# B&R Automation Studio project mapp6d_SampleProject
Automation Studio 4.10.2.37; technology packages: mapp6D 1.1.7924

## Configuration Config1

CPU X20CP3586, AutomationRuntime B4.91, Build 4.1.2, Safety 0.0, Vc V4.72.3

### Task classes (Cpu.sw)
```
Cyclic#4:
  Program <- Program.prg
Libraries: McAcp6D, McBase, AsMath
```

### Hardware
```
8YFLM01.0000.00I-1 : 8YFLM01.0000.00I-1 v0.0.0.1  [PLK1 -> X20CP3586.IF3 (NodeNumber=16) [Cable Type=PowerlinkCable, Length=10, Version=1.0.0.3]]
  Supervision = off
X20CP3586 : X20CP3586 v1.9.0.0
  Connector IF2:
    ActivateDevice = 1
    Mode = Manual
    InternetAddress = 192.168.10.7
    SubnetMask = 255.255.255.0
    ActivateSnmp = 2
  Connector IF3:
    CycleTime = 1000
  ConfigurationID = mapp6d_SampleProject_Config1
  TimerDeviceType = EPLX2X
  TimerDevice = X20CP3586.IF3
  TaskClassIdleTime = 2000
  Cyclic1Duration = 1000
  Cyclic1Tolerance = 0
  Cyclic3Duration = 52000
  Cyclic3Tolerance = 52000
  Cyclic5Duration = 198000
  Cyclic5Tolerance = 198000
  Cyclic7Duration = 1002000
  Cyclic7Tolerance = 1002000
  FileDevice1
  FileDeviceName1 = 6DData
  FileDevicePath1 = C:\
  FtpUser1
  FtpUsername1 = admin
  FtpUserPassword1 = lR/ROkjEB6ZsaZw8IVX3MB+yAH7U94gbA110ofjiao0=  // admin
  FtpUserSalt1 = rhukc7YS
  FTPAccessRight1 = 0
  FTPdevice1 = ALL
```

### IoMap.iom - X20CP3586/IoMap.iom
```iecst
VAR_CONFIG
	Cyclic#1.::FBin.Array[0] AT %IW."8YFLM01.0000.00I-1".EPL_FB_IN_0_I2007_S01;
	Cyclic#1.::FBin.Array[1] AT %IW."8YFLM01.0000.00I-1".EPL_FB_IN_1_I2007_S02;
	Cyclic#1.::FBin.Array[10] AT %IW."8YFLM01.0000.00I-1".EPL_FB_IN_10_I2007_S0B;
	Cyclic#1.::FBin.Array[100] AT %IW."8YFLM01.0000.00I-1".EPL_FB_IN_100_I2007_S65;
	Cyclic#1.::FBin.Array[101] AT %IW."8YFLM01.0000.00I-1".EPL_FB_IN_101_I2007_S66;
	Cyclic#1.::FBin.Array[102] AT %IW."8YFLM01.0000.00I-1".EPL_FB_IN_102_I2007_S67;
	Cyclic#1.::FBin.Array[103] AT %IW."8YFLM01.0000.00I-1".EPL_FB_IN_103_I2007_S68;
	Cyclic#1.::FBin.Array[104] AT %IW."8YFLM01.0000.00I-1".EPL_FB_IN_104_I2007_S69;
	Cyclic#1.::FBin.Array[105] AT %IW."8YFLM01.0000.00I-1".EPL_FB_IN_105_I2007_S6A;
	Cyclic#1.::FBin.Array[106] AT %IW."8YFLM01.0000.00I-1".EPL_FB_IN_106_I2007_S6B;
	Cyclic#1.::FBin.Array[107] AT %IW."8YFLM01.0000.00I-1".EPL_FB_IN_107_I2007_S6C;
	Cyclic#1.::FBin.Array[108] AT %IW."8YFLM01.0000.00I-1".EPL_FB_IN_108_I2007_S6D;
	Cyclic#1.::FBin.Array[109] AT %IW."8YFLM01.0000.00I-1".EPL_FB_IN_109_I2007_S6E;
	Cyclic#1.::FBin.Array[11] AT %IW."8YFLM01.0000.00I-1".EPL_FB_IN_11_I2007_S0C;
	Cyclic#1.::FBin.Array[110] AT %IW."8YFLM01.0000.00I-1".EPL_FB_IN_110_I2007_S6F;
	Cyclic#1.::FBin.Array[111] AT %IW."8YFLM01.0000.00I-1".EPL_FB_IN_111_I2007_S70;
	Cyclic#1.::FBin.Array[112] AT %IW."8YFLM01.0000.00I-1".EPL_FB_IN_112_I2007_S71;
	Cyclic#1.::FBin.Array[113] AT %IW."8YFLM01.0000.00I-1".EPL_FB_IN_113_I2007_S72;
	Cyclic#1.::FBin.Array[114] AT %IW."8YFLM01.0000.00I-1".EPL_FB_IN_114_I2007_S73;
	Cyclic#1.::FBin.Array[115] AT %IW."8YFLM01.0000.00I-1".EPL_FB_IN_115_I2007_S74;
	Cyclic#1.::FBin.Array[116] AT %IW."8YFLM01.0000.00I-1".EPL_FB_IN_116_I2007_S75;
	Cyclic#1.::FBin.Array[117] AT %IW."8YFLM01.0000.00I-1".EPL_FB_IN_117_I2007_S76;
	Cyclic#1.::FBin.Array[118] AT %IW."8YFLM01.0000.00I-1".EPL_FB_IN_118_I2007_S77;
	Cyclic#1.::FBin.Array[119] AT %IW."8YFLM01.0000.00I-1".EPL_FB_IN_119_I2007_S78;
	Cyclic#1.::FBin.Array[12] AT %IW."8YFLM01.0000.00I-1".EPL_FB_IN_12_I2007_S0D;
	Cyclic#1.::FBin.Array[120] AT %IW."8YFLM01.0000.00I-1".EPL_FB_IN_120_I2007_S79;
	Cyclic#1.::FBin.Array[121] AT %IW."8YFLM01.0000.00I-1".EPL_FB_IN_121_I2007_S7A;
	Cyclic#1.::FBin.Array[122] AT %IW."8YFLM01.0000.00I-1".EPL_FB_IN_122_I2007_S7B;
	Cyclic#1.::FBin.Array[123] AT %IW."8YFLM01.0000.00I-1".EPL_FB_IN_123_I2007_S7C;
	Cyclic#1.::FBin.Array[124] AT %IW."8YFLM01.0000.00I-1".EPL_FB_IN_124_I2007_S7D;
	Cyclic#1.::FBin.Array[125] AT %IW."8YFLM01.0000.00I-1".EPL_FB_IN_125_I2007_S7E;
	Cyclic#1.::FBin.Array[126] AT %IW."8YFLM01.0000.00I-1".EPL_FB_IN_126_I2007_S7F;
	Cyclic#1.::FBin.Array[127] AT %IW."8YFLM01.0000.00I-1".EPL_FB_IN_127_I2007_S80;
	Cyclic#1.::FBin.Array[128] AT %IW."8YFLM01.0000.00I-1".EPL_FB_IN_128_I2007_S81;
	Cyclic#1.::FBin.Array[129] AT %IW."8YFLM01.0000.00I-1".EPL_FB_IN_129_I2007_S82;
	Cyclic#1.::FBin.Array[13] AT %IW."8YFLM01.0000.00I-1".EPL_FB_IN_13_I2007_S0E;
	Cyclic#1.::FBin.Array[130] AT %IW."8YFLM01.0000.00I-1".EPL_FB_IN_130_I2007_S83;
	Cyclic#1.::FBin.Array[131] AT %IW."8YFLM01.0000.00I-1".EPL_FB_IN_131_I2007_S84;
	Cyclic#1.::FBin.Array[132] AT %IW."8YFLM01.0000.00I-1".EPL_FB_IN_132_I2007_S85;
	Cyclic#1.::FBin.Array[133] AT %IW."8YFLM01.0000.00I-1".EPL_FB_IN_133_I2007_S86;
	Cyclic#1.::FBin.Array[134] AT %IW."8YFLM01.0000.00I-1".EPL_FB_IN_134_I2007_S87;
	Cyclic#1.::FBin.Array[135] AT %IW."8YFLM01.0000.00I-1".EPL_FB_IN_135_I2007_S88;
	Cyclic#1.::FBin.Array[136] AT %IW."8YFLM01.0000.00I-1".EPL_FB_IN_136_I2007_S89;
	Cyclic#1.::FBin.Array[137] AT %IW."8YFLM01.0000.00I-1".EPL_FB_IN_137_I2007_S8A;
	Cyclic#1.::FBin.Array[138] AT %IW."8YFLM01.0000.00I-1".EPL_FB_IN_138_I2007_S8B;
	Cyclic#1.::FBin.Array[139] AT %IW."8YFLM01.0000.00I-1".EPL_FB_IN_139_I2007_S8C;
	Cyclic#1.::FBin.Array[14] AT %IW."8YFLM01.0000.00I-1".EPL_FB_IN_14_I2007_S0F;
	Cyclic#1.::FBin.Array[140] AT %IW."8YFLM01.0000.00I-1".EPL_FB_IN_140_I2007_S8D;
	Cyclic#1.::FBin.Array[141] AT %IW."8YFLM01.0000.00I-1".EPL_FB_IN_141_I2007_S8E;
	Cyclic#1.::FBin.Array[142] AT %IW."8YFLM01.0000.00I-1".EPL_FB_IN_142_I2007_S8F;
	Cyclic#1.::FBin.Array[143] AT %IW."8YFLM01.0000.00I-1".EPL_FB_IN_143_I2007_S90;
	Cyclic#1.::FBin.Array[144] AT %IW."8YFLM01.0000.00I-1".EPL_FB_IN_144_I2007_S91;
	Cyclic#1.::FBin.Array[145] AT %IW."8YFLM01.0000.00I-1".EPL_FB_IN_145_I2007_S92;
	Cyclic#1.::FBin.Array[146] AT %IW."8YFLM01.0000.00I-1".EPL_FB_IN_146_I2007_S93;
	Cyclic#1.::FBin.Array[147] AT %IW."8YFLM01.0000.00I-1".EPL_FB_IN_147_I2007_S94;
	Cyclic#1.::FBin.Array[148] AT %IW."8YFLM01.0000.00I-1".EPL_FB_IN_148_I2007_S95;
	Cyclic#1.::FBin.Array[149] AT %IW."8YFLM01.0000.00I-1".EPL_FB_IN_149_I2007_S96;
	Cyclic#1.::FBin.Array[15] AT %IW."8YFLM01.0000.00I-1".EPL_FB_IN_15_I2007_S10;
	Cyclic#1.::FBin.Array[150] AT %IW."8YFLM01.0000.00I-1".EPL_FB_IN_150_I2007_S97;
	Cyclic#1.::FBin.Array[151] AT %IW."8YFLM01.0000.00I-1".EPL_FB_IN_151_I2007_S98;
	Cyclic#1.::FBin.Array[152] AT %IW."8YFLM01.0000.00I-1".EPL_FB_IN_152_I2007_S99;
	Cyclic#1.::FBin.Array[153] AT %IW."8YFLM01.0000.00I-1".EPL_FB_IN_153_I2007_S9A;
	Cyclic#1.::FBin.Array[154] AT %IW."8YFLM01.0000.00I-1".EPL_FB_IN_154_I2007_S9B;
	Cyclic#1.::FBin.Array[155] AT %IW."8YFLM01.0000.00I-1".EPL_FB_IN_155_I2007_S9C;
	Cyclic#1.::FBin.Array[156] AT %IW."8YFLM01.0000.00I-1".EPL_FB_IN_156_I2007_S9D;
	Cyclic#1.::FBin.Array[157] AT %IW."8YFLM01.0000.00I-1".EPL_FB_IN_157_I2007_S9E;
	Cyclic#1.::FBin.Array[158] AT %IW."8YFLM01.0000.00I-1".EPL_FB_IN_158_I2007_S9F;
	Cyclic#1.::FBin.Array[159] AT %IW."8YFLM01.0000.00I-1".EPL_FB_IN_159_I2007_SA0;
	Cyclic#1.::FBin.Array[16] AT %IW."8YFLM01.0000.00I-1".EPL_FB_IN_16_I2007_S11;
	Cyclic#1.::FBin.Array[160] AT %IW."8YFLM01.0000.00I-1".EPL_FB_IN_160_I2007_SA1;
	Cyclic#1.::FBin.Array[161] AT %IW."8YFLM01.0000.00I-1".EPL_FB_IN_161_I2007_SA2;
	Cyclic#1.::FBin.Array[162] AT %IW."8YFLM01.0000.00I-1".EPL_FB_IN_162_I2007_SA3;
	Cyclic#1.::FBin.Array[163] AT %IW."8YFLM01.0000.00I-1".EPL_FB_IN_163_I2007_SA4;
	Cyclic#1.::FBin.Array[164] AT %IW."8YFLM01.0000.00I-1".EPL_FB_IN_164_I2007_SA5;
	Cyclic#1.::FBin.Array[165] AT %IW."8YFLM01.0000.00I-1".EPL_FB_IN_165_I2007_SA6;
	Cyclic#1.::FBin.Array[166] AT %IW."8YFLM01.0000.00I-1".EPL_FB_IN_166_I2007_SA7;
	Cyclic#1.::FBin.Array[167] AT %IW."8YFLM01.0000.00I-1".EPL_FB_IN_167_I2007_SA8;
	Cyclic#1.::FBin.Array[168] AT %IW."8YFLM01.0000.00I-1".EPL_FB_IN_168_I2007_SA9;
	Cyclic#1.::FBin.Array[169] AT %IW."8YFLM01.0000.00I-1".EPL_FB_IN_169_I2007_SAA;
	Cyclic#1.::FBin.Array[17] AT %IW."8YFLM01.0000.00I-1".EPL_FB_IN_17_I2007_S12;
	Cyclic#1.::FBin.Array[170] AT %IW."8YFLM01.0000.00I-1".EPL_FB_IN_170_I2007_SAB;
	Cyclic#1.::FBin.Array[171] AT %IW."8YFLM01.0000.00I-1".EPL_FB_IN_171_I2007_SAC;
	Cyclic#1.::FBin.Array[172] AT %IW."8YFLM01.0000.00I-1".EPL_FB_IN_172_I2007_SAD;
	Cyclic#1.::FBin.Array[173] AT %IW."8YFLM01.0000.00I-1".EPL_FB_IN_173_I2007_SAE;
	Cyclic#1.::FBin.Array[174] AT %IW."8YFLM01.0000.00I-1".EPL_FB_IN_174_I2007_SAF;
	Cyclic#1.::FBin.Array[175] AT %IW."8YFLM01.0000.00I-1".EPL_FB_IN_175_I2007_SB0;
	Cyclic#1.::FBin.Array[176] AT %IW."8YFLM01.0000.00I-1".EPL_FB_IN_176_I2007_SB1;
	Cyclic#1.::FBin.Array[177] AT %IW."8YFLM01.0000.00I-1".EPL_FB_IN_177_I2007_SB2;
	Cyclic#1.::FBin.Array[178] AT %IW."8YFLM01.0000.00I-1".EPL_FB_IN_178_I2007_SB3;
	Cyclic#1.::FBin.Array[179] AT %IW."8YFLM01.0000.00I-1".EPL_FB_IN_179_I2007_SB4;
	Cyclic#1.::FBin.Array[18] AT %IW."8YFLM01.0000.00I-1".EPL_FB_IN_18_I2007_S13;
	Cyclic#1.::FBin.Array[180] AT %IW."8YFLM01.0000.00I-1".EPL_FB_IN_180_I2007_SB5;
	Cyclic#1.::FBin.Array[181] AT %IW."8YFLM01.0000.00I-1".EPL_FB_IN_181_I2007_SB6;
	Cyclic#1.::FBin.Array[182] AT %IW."8YFLM01.0000.00I-1".EPL_FB_IN_182_I2007_SB7;
	Cyclic#1.::FBin.Array[183] AT %IW."8YFLM01.0000.00I-1".EPL_FB_IN_183_I2007_SB8;
	Cyclic#1.::FBin.Array[184] AT %IW."8YFLM01.0000.00I-1".EPL_FB_IN_184_I2007_SB9;
	Cyclic#1.::FBin.Array[185] AT %IW."8YFLM01.0000.00I-1".EPL_FB_IN_185_I2007_SBA;
	Cyclic#1.::FBin.Array[186] AT %IW."8YFLM01.0000.00I-1".EPL_FB_IN_186_I2007_SBB;
	Cyclic#1.::FBin.Array[187] AT %IW."8YFLM01.0000.00I-1".EPL_FB_IN_187_I2007_SBC;
	Cyclic#1.::FBin.Array[188] AT %IW."8YFLM01.0000.00I-1".EPL_FB_IN_188_I2007_SBD;
	Cyclic#1.::FBin.Array[189] AT %IW."8YFLM01.0000.00I-1".EPL_FB_IN_189_I2007_SBE;
	Cyclic#1.::FBin.Array[19] AT %IW."8YFLM01.0000.00I-1".EPL_FB_IN_19_I2007_S14;
	Cyclic#1.::FBin.Array[190] AT %IW."8YFLM01.0000.00I-1".EPL_FB_IN_190_I2007_SBF;
	Cyclic#1.::FBin.Array[191] AT %IW."8YFLM01.0000.00I-1".EPL_FB_IN_191_I2007_SC0;
	Cyclic#1.::FBin.Array[192] AT %IW."8YFLM01.0000.00I-1".EPL_FB_IN_192_I2007_SC1;
	Cyclic#1.::FBin.Array[193] AT %IW."8YFLM01.0000.00I-1".EPL_FB_IN_193_I2007_SC2;
	Cyclic#1.::FBin.Array[194] AT %IW."8YFLM01.0000.00I-1".EPL_FB_IN_194_I2007_SC3;
	Cyclic#1.::FBin.Array[195] AT %IW."8YFLM01.0000.00I-1".EPL_FB_IN_195_I2007_SC4;
	Cyclic#1.::FBin.Array[196] AT %IW."8YFLM01.0000.00I-1".EPL_FB_IN_196_I2007_SC5;
	Cyclic#1.::FBin.Array[197] AT %IW."8YFLM01.0000.00I-1".EPL_FB_IN_197_I2007_SC6;
	Cyclic#1.::FBin.Array[198] AT %IW."8YFLM01.0000.00I-1".EPL_FB_IN_198_I2007_SC7;
	Cyclic#1.::FBin.Array[199] AT %IW."8YFLM01.0000.00I-1".EPL_FB_IN_199_I2007_SC8;
	Cyclic#1.::FBin.Array[2] AT %IW."8YFLM01.0000.00I-1".EPL_FB_IN_2_I2007_S03;
	Cyclic#1.::FBin.Array[20] AT %IW."8YFLM01.0000.00I-1".EPL_FB_IN_20_I2007_S15;
	Cyclic#1.::FBin.Array[21] AT %IW."8YFLM01.0000.00I-1".EPL_FB_IN_21_I2007_S16;
	Cyclic#1.::FBin.Array[22] AT %IW."8YFLM01.0000.00I-1".EPL_FB_IN_22_I2007_S17;
	Cyclic#1.::FBin.Array[23] AT %IW."8YFLM01.0000.00I-1".EPL_FB_IN_23_I2007_S18;
	Cyclic#1.::FBin.Array[24] AT %IW."8YFLM01.0000.00I-1".EPL_FB_IN_24_I2007_S19;
	Cyclic#1.::FBin.Array[25] AT %IW."8YFLM01.0000.00I-1".EPL_FB_IN_25_I2007_S1A;
	Cyclic#1.::FBin.Array[26] AT %IW."8YFLM01.0000.00I-1".EPL_FB_IN_26_I2007_S1B;
	Cyclic#1.::FBin.Array[27] AT %IW."8YFLM01.0000.00I-1".EPL_FB_IN_27_I2007_S1C;
	Cyclic#1.::FBin.Array[28] AT %IW."8YFLM01.0000.00I-1".EPL_FB_IN_28_I2007_S1D;
	Cyclic#1.::FBin.Array[29] AT %IW."8YFLM01.0000.00I-1".EPL_FB_IN_29_I2007_S1E;
	Cyclic#1.::FBin.Array[3] AT %IW."8YFLM01.0000.00I-1".EPL_FB_IN_3_I2007_S04;
	Cyclic#1.::FBin.Array[30] AT %IW."8YFLM01.0000.00I-1".EPL_FB_IN_30_I2007_S1F;
	Cyclic#1.::FBin.Array[31] AT %IW."8YFLM01.0000.00I-1".EPL_FB_IN_31_I2007_S20;
	Cyclic#1.::FBin.Array[32] AT %IW."8YFLM01.0000.00I-1".EPL_FB_IN_32_I2007_S21;
	Cyclic#1.::FBin.Array[33] AT %IW."8YFLM01.0000.00I-1".EPL_FB_IN_33_I2007_S22;
	Cyclic#1.::FBin.Array[34] AT %IW."8YFLM01.0000.00I-1".EPL_FB_IN_34_I2007_S23;
	Cyclic#1.::FBin.Array[35] AT %IW."8YFLM01.0000.00I-1".EPL_FB_IN_35_I2007_S24;
	Cyclic#1.::FBin.Array[36] AT %IW."8YFLM01.0000.00I-1".EPL_FB_IN_36_I2007_S25;
	Cyclic#1.::FBin.Array[37] AT %IW."8YFLM01.0000.00I-1".EPL_FB_IN_37_I2007_S26;
	Cyclic#1.::FBin.Array[38] AT %IW."8YFLM01.0000.00I-1".EPL_FB_IN_38_I2007_S27;
	Cyclic#1.::FBin.Array[39] AT %IW."8YFLM01.0000.00I-1".EPL_FB_IN_39_I2007_S28;
	Cyclic#1.::FBin.Array[4] AT %IW."8YFLM01.0000.00I-1".EPL_FB_IN_4_I2007_S05;
	Cyclic#1.::FBin.Array[40] AT %IW."8YFLM01.0000.00I-1".EPL_FB_IN_40_I2007_S29;
	Cyclic#1.::FBin.Array[41] AT %IW."8YFLM01.0000.00I-1".EPL_FB_IN_41_I2007_S2A;
	Cyclic#1.::FBin.Array[42] AT %IW."8YFLM01.0000.00I-1".EPL_FB_IN_42_I2007_S2B;
	Cyclic#1.::FBin.Array[43] AT %IW."8YFLM01.0000.00I-1".EPL_FB_IN_43_I2007_S2C;
	Cyclic#1.::FBin.Array[44] AT %IW."8YFLM01.0000.00I-1".EPL_FB_IN_44_I2007_S2D;
	Cyclic#1.::FBin.Array[45] AT %IW."8YFLM01.0000.00I-1".EPL_FB_IN_45_I2007_S2E;
	Cyclic#1.::FBin.Array[46] AT %IW."8YFLM01.0000.00I-1".EPL_FB_IN_46_I2007_S2F;
	Cyclic#1.::FBin.Array[47] AT %IW."8YFLM01.0000.00I-1".EPL_FB_IN_47_I2007_S30;
	Cyclic#1.::FBin.Array[48] AT %IW."8YFLM01.0000.00I-1".EPL_FB_IN_48_I2007_S31;
	Cyclic#1.::FBin.Array[49] AT %IW."8YFLM01.0000.00I-1".EPL_FB_IN_49_I2007_S32;
	Cyclic#1.::FBin.Array[5] AT %IW."8YFLM01.0000.00I-1".EPL_FB_IN_5_I2007_S06;
	Cyclic#1.::FBin.Array[50] AT %IW."8YFLM01.0000.00I-1".EPL_FB_IN_50_I2007_S33;
	Cyclic#1.::FBin.Array[51] AT %IW."8YFLM01.0000.00I-1".EPL_FB_IN_51_I2007_S34;
	Cyclic#1.::FBin.Array[52] AT %IW."8YFLM01.0000.00I-1".EPL_FB_IN_52_I2007_S35;
	Cyclic#1.::FBin.Array[53] AT %IW."8YFLM01.0000.00I-1".EPL_FB_IN_53_I2007_S36;
	Cyclic#1.::FBin.Array[54] AT %IW."8YFLM01.0000.00I-1".EPL_FB_IN_54_I2007_S37;
	Cyclic#1.::FBin.Array[55] AT %IW."8YFLM01.0000.00I-1".EPL_FB_IN_55_I2007_S38;
	Cyclic#1.::FBin.Array[56] AT %IW."8YFLM01.0000.00I-1".EPL_FB_IN_56_I2007_S39;
	Cyclic#1.::FBin.Array[57] AT %IW."8YFLM01.0000.00I-1".EPL_FB_IN_57_I2007_S3A;
	Cyclic#1.::FBin.Array[58] AT %IW."8YFLM01.0000.00I-1".EPL_FB_IN_58_I2007_S3B;
	Cyclic#1.::FBin.Array[59] AT %IW."8YFLM01.0000.00I-1".EPL_FB_IN_59_I2007_S3C;
	Cyclic#1.::FBin.Array[6] AT %IW."8YFLM01.0000.00I-1".EPL_FB_IN_6_I2007_S07;
	Cyclic#1.::FBin.Array[60] AT %IW."8YFLM01.0000.00I-1".EPL_FB_IN_60_I2007_S3D;
	Cyclic#1.::FBin.Array[61] AT %IW."8YFLM01.0000.00I-1".EPL_FB_IN_61_I2007_S3E;
	Cyclic#1.::FBin.Array[62] AT %IW."8YFLM01.0000.00I-1".EPL_FB_IN_62_I2007_S3F;
	Cyclic#1.::FBin.Array[63] AT %IW."8YFLM01.0000.00I-1".EPL_FB_IN_63_I2007_S40;
	Cyclic#1.::FBin.Array[64] AT %IW."8YFLM01.0000.00I-1".EPL_FB_IN_64_I2007_S41;
	Cyclic#1.::FBin.Array[65] AT %IW."8YFLM01.0000.00I-1".EPL_FB_IN_65_I2007_S42;
	Cyclic#1.::FBin.Array[66] AT %IW."8YFLM01.0000.00I-1".EPL_FB_IN_66_I2007_S43;
	Cyclic#1.::FBin.Array[67] AT %IW."8YFLM01.0000.00I-1".EPL_FB_IN_67_I2007_S44;
	Cyclic#1.::FBin.Array[68] AT %IW."8YFLM01.0000.00I-1".EPL_FB_IN_68_I2007_S45;
	Cyclic#1.::FBin.Array[69] AT %IW."8YFLM01.0000.00I-1".EPL_FB_IN_69_I2007_S46;
	Cyclic#1.::FBin.Array[7] AT %IW."8YFLM01.0000.00I-1".EPL_FB_IN_7_I2007_S08;
	Cyclic#1.::FBin.Array[70] AT %IW."8YFLM01.0000.00I-1".EPL_FB_IN_70_I2007_S47;
	Cyclic#1.::FBin.Array[71] AT %IW."8YFLM01.0000.00I-1".EPL_FB_IN_71_I2007_S48;
	Cyclic#1.::FBin.Array[72] AT %IW."8YFLM01.0000.00I-1".EPL_FB_IN_72_I2007_S49;
	Cyclic#1.::FBin.Array[73] AT %IW."8YFLM01.0000.00I-1".EPL_FB_IN_73_I2007_S4A;
	Cyclic#1.::FBin.Array[74] AT %IW."8YFLM01.0000.00I-1".EPL_FB_IN_74_I2007_S4B;
	Cyclic#1.::FBin.Array[75] AT %IW."8YFLM01.0000.00I-1".EPL_FB_IN_75_I2007_S4C;
	Cyclic#1.::FBin.Array[76] AT %IW."8YFLM01.0000.00I-1".EPL_FB_IN_76_I2007_S4D;
	Cyclic#1.::FBin.Array[77] AT %IW."8YFLM01.0000.00I-1".EPL_FB_IN_77_I2007_S4E;
	Cyclic#1.::FBin.Array[78] AT %IW."8YFLM01.0000.00I-1".EPL_FB_IN_78_I2007_S4F;
	Cyclic#1.::FBin.Array[79] AT %IW."8YFLM01.0000.00I-1".EPL_FB_IN_79_I2007_S50;
	Cyclic#1.::FBin.Array[8] AT %IW."8YFLM01.0000.00I-1".EPL_FB_IN_8_I2007_S09;
	Cyclic#1.::FBin.Array[80] AT %IW."8YFLM01.0000.00I-1".EPL_FB_IN_80_I2007_S51;
	Cyclic#1.::FBin.Array[81] AT %IW."8YFLM01.0000.00I-1".EPL_FB_IN_81_I2007_S52;
	Cyclic#1.::FBin.Array[82] AT %IW."8YFLM01.0000.00I-1".EPL_FB_IN_82_I2007_S53;
	Cyclic#1.::FBin.Array[83] AT %IW."8YFLM01.0000.00I-1".EPL_FB_IN_83_I2007_S54;
	Cyclic#1.::FBin.Array[84] AT %IW."8YFLM01.0000.00I-1".EPL_FB_IN_84_I2007_S55;
	Cyclic#1.::FBin.Array[85] AT %IW."8YFLM01.0000.00I-1".EPL_FB_IN_85_I2007_S56;
	Cyclic#1.::FBin.Array[86] AT %IW."8YFLM01.0000.00I-1".EPL_FB_IN_86_I2007_S57;
	Cyclic#1.::FBin.Array[87] AT %IW."8YFLM01.0000.00I-1".EPL_FB_IN_87_I2007_S58;
	Cyclic#1.::FBin.Array[88] AT %IW."8YFLM01.0000.00I-1".EPL_FB_IN_88_I2007_S59;
	Cyclic#1.::FBin.Array[89] AT %IW."8YFLM01.0000.00I-1".EPL_FB_IN_89_I2007_S5A;
	Cyclic#1.::FBin.Array[9] AT %IW."8YFLM01.0000.00I-1".EPL_FB_IN_9_I2007_S0A;
	Cyclic#1.::FBin.Array[90] AT %IW."8YFLM01.0000.00I-1".EPL_FB_IN_90_I2007_S5B;
	Cyclic#1.::FBin.Array[91] AT %IW."8YFLM01.0000.00I-1".EPL_FB_IN_91_I2007_S5C;
	Cyclic#1.::FBin.Array[92] AT %IW."8YFLM01.0000.00I-1".EPL_FB_IN_92_I2007_S5D;
	Cyclic#1.::FBin.Array[93] AT %IW."8YFLM01.0000.00I-1".EPL_FB_IN_93_I2007_S5E;
	Cyclic#1.::FBin.Array[94] AT %IW."8YFLM01.0000.00I-1".EPL_FB_IN_94_I2007_S5F;
	Cyclic#1.::FBin.Array[95] AT %IW."8YFLM01.0000.00I-1".EPL_FB_IN_95_I2007_S60;
	Cyclic#1.::FBin.Array[96] AT %IW."8YFLM01.0000.00I-1".EPL_FB_IN_96_I2007_S61;
	Cyclic#1.::FBin.Array[97] AT %IW."8YFLM01.0000.00I-1".EPL_FB_IN_97_I2007_S62;
	Cyclic#1.::FBin.Array[98] AT %IW."8YFLM01.0000.00I-1".EPL_FB_IN_98_I2007_S63;
	Cyclic#1.::FBin.Array[99] AT %IW."8YFLM01.0000.00I-1".EPL_FB_IN_99_I2007_S64;
	Cyclic#1.::FBout.Array[0] AT %QW."8YFLM01.0000.00I-1".EPL_FB_OUT_0_I2008_S01Out;
	Cyclic#1.::FBout.Array[1] AT %QW."8YFLM01.0000.00I-1".EPL_FB_OUT_1_I2008_S02Out;
	Cyclic#1.::FBout.Array[10] AT %QW."8YFLM01.0000.00I-1".EPL_FB_OUT_10_I2008_S0BOut;
	Cyclic#1.::FBout.Array[100] AT %QW."8YFLM01.0000.00I-1".EPL_FB_OUT_100_I2008_S65Out;
	Cyclic#1.::FBout.Array[101] AT %QW."8YFLM01.0000.00I-1".EPL_FB_OUT_101_I2008_S66Out;
	Cyclic#1.::FBout.Array[102] AT %QW."8YFLM01.0000.00I-1".EPL_FB_OUT_102_I2008_S67Out;
	Cyclic#1.::FBout.Array[103] AT %QW."8YFLM01.0000.00I-1".EPL_FB_OUT_103_I2008_S68Out;
	Cyclic#1.::FBout.Array[104] AT %QW."8YFLM01.0000.00I-1".EPL_FB_OUT_104_I2008_S69Out;
	Cyclic#1.::FBout.Array[105] AT %QW."8YFLM01.0000.00I-1".EPL_FB_OUT_105_I2008_S6AOut;
	Cyclic#1.::FBout.Array[106] AT %QW."8YFLM01.0000.00I-1".EPL_FB_OUT_106_I2008_S6BOut;
	Cyclic#1.::FBout.Array[107] AT %QW."8YFLM01.0000.00I-1".EPL_FB_OUT_107_I2008_S6COut;
	Cyclic#1.::FBout.Array[108] AT %QW."8YFLM01.0000.00I-1".EPL_FB_OUT_108_I2008_S6DOut;
	Cyclic#1.::FBout.Array[109] AT %QW."8YFLM01.0000.00I-1".EPL_FB_OUT_109_I2008_S6EOut;
	Cyclic#1.::FBout.Array[11] AT %QW."8YFLM01.0000.00I-1".EPL_FB_OUT_11_I2008_S0COut;
	Cyclic#1.::FBout.Array[110] AT %QW."8YFLM01.0000.00I-1".EPL_FB_OUT_110_I2008_S6FOut;
	Cyclic#1.::FBout.Array[111] AT %QW."8YFLM01.0000.00I-1".EPL_FB_OUT_111_I2008_S70Out;
	Cyclic#1.::FBout.Array[112] AT %QW."8YFLM01.0000.00I-1".EPL_FB_OUT_112_I2008_S71Out;
	Cyclic#1.::FBout.Array[113] AT %QW."8YFLM01.0000.00I-1".EPL_FB_OUT_113_I2008_S72Out;
	Cyclic#1.::FBout.Array[114] AT %QW."8YFLM01.0000.00I-1".EPL_FB_OUT_114_I2008_S73Out;
	Cyclic#1.::FBout.Array[115] AT %QW."8YFLM01.0000.00I-1".EPL_FB_OUT_115_I2008_S74Out;
	Cyclic#1.::FBout.Array[116] AT %QW."8YFLM01.0000.00I-1".EPL_FB_OUT_116_I2008_S75Out;
	Cyclic#1.::FBout.Array[117] AT %QW."8YFLM01.0000.00I-1".EPL_FB_OUT_117_I2008_S76Out;
	Cyclic#1.::FBout.Array[118] AT %QW."8YFLM01.0000.00I-1".EPL_FB_OUT_118_I2008_S77Out;
	Cyclic#1.::FBout.Array[119] AT %QW."8YFLM01.0000.00I-1".EPL_FB_OUT_119_I2008_S78Out;
	Cyclic#1.::FBout.Array[12] AT %QW."8YFLM01.0000.00I-1".EPL_FB_OUT_12_I2008_S0DOut;
	Cyclic#1.::FBout.Array[120] AT %QW."8YFLM01.0000.00I-1".EPL_FB_OUT_120_I2008_S79Out;
	Cyclic#1.::FBout.Array[121] AT %QW."8YFLM01.0000.00I-1".EPL_FB_OUT_121_I2008_S7AOut;
	Cyclic#1.::FBout.Array[122] AT %QW."8YFLM01.0000.00I-1".EPL_FB_OUT_122_I2008_S7BOut;
	Cyclic#1.::FBout.Array[123] AT %QW."8YFLM01.0000.00I-1".EPL_FB_OUT_123_I2008_S7COut;
	Cyclic#1.::FBout.Array[124] AT %QW."8YFLM01.0000.00I-1".EPL_FB_OUT_124_I2008_S7DOut;
	Cyclic#1.::FBout.Array[125] AT %QW."8YFLM01.0000.00I-1".EPL_FB_OUT_125_I2008_S7EOut;
	Cyclic#1.::FBout.Array[126] AT %QW."8YFLM01.0000.00I-1".EPL_FB_OUT_126_I2008_S7FOut;
	Cyclic#1.::FBout.Array[127] AT %QW."8YFLM01.0000.00I-1".EPL_FB_OUT_127_I2008_S80Out;
	Cyclic#1.::FBout.Array[128] AT %QW."8YFLM01.0000.00I-1".EPL_FB_OUT_128_I2008_S81Out;
	Cyclic#1.::FBout.Array[129] AT %QW."8YFLM01.0000.00I-1".EPL_FB_OUT_129_I2008_S82Out;
	Cyclic#1.::FBout.Array[13] AT %QW."8YFLM01.0000.00I-1".EPL_FB_OUT_13_I2008_S0EOut;
	Cyclic#1.::FBout.Array[130] AT %QW."8YFLM01.0000.00I-1".EPL_FB_OUT_130_I2008_S83Out;
	Cyclic#1.::FBout.Array[131] AT %QW."8YFLM01.0000.00I-1".EPL_FB_OUT_131_I2008_S84Out;
	Cyclic#1.::FBout.Array[132] AT %QW."8YFLM01.0000.00I-1".EPL_FB_OUT_132_I2008_S85Out;
	Cyclic#1.::FBout.Array[133] AT %QW."8YFLM01.0000.00I-1".EPL_FB_OUT_133_I2008_S86Out;
	Cyclic#1.::FBout.Array[134] AT %QW."8YFLM01.0000.00I-1".EPL_FB_OUT_134_I2008_S87Out;
	Cyclic#1.::FBout.Array[135] AT %QW."8YFLM01.0000.00I-1".EPL_FB_OUT_135_I2008_S88Out;
	Cyclic#1.::FBout.Array[136] AT %QW."8YFLM01.0000.00I-1".EPL_FB_OUT_136_I2008_S89Out;
	Cyclic#1.::FBout.Array[137] AT %QW."8YFLM01.0000.00I-1".EPL_FB_OUT_137_I2008_S8AOut;
	Cyclic#1.::FBout.Array[138] AT %QW."8YFLM01.0000.00I-1".EPL_FB_OUT_138_I2008_S8BOut;
	Cyclic#1.::FBout.Array[139] AT %QW."8YFLM01.0000.00I-1".EPL_FB_OUT_139_I2008_S8COut;
	Cyclic#1.::FBout.Array[14] AT %QW."8YFLM01.0000.00I-1".EPL_FB_OUT_14_I2008_S0FOut;
	Cyclic#1.::FBout.Array[140] AT %QW."8YFLM01.0000.00I-1".EPL_FB_OUT_140_I2008_S8DOut;
	Cyclic#1.::FBout.Array[141] AT %QW."8YFLM01.0000.00I-1".EPL_FB_OUT_141_I2008_S8EOut;
	Cyclic#1.::FBout.Array[142] AT %QW."8YFLM01.0000.00I-1".EPL_FB_OUT_142_I2008_S8FOut;
	Cyclic#1.::FBout.Array[143] AT %QW."8YFLM01.0000.00I-1".EPL_FB_OUT_143_I2008_S90Out;
	Cyclic#1.::FBout.Array[144] AT %QW."8YFLM01.0000.00I-1".EPL_FB_OUT_144_I2008_S91Out;
	Cyclic#1.::FBout.Array[145] AT %QW."8YFLM01.0000.00I-1".EPL_FB_OUT_145_I2008_S92Out;
	Cyclic#1.::FBout.Array[146] AT %QW."8YFLM01.0000.00I-1".EPL_FB_OUT_146_I2008_S93Out;
	Cyclic#1.::FBout.Array[147] AT %QW."8YFLM01.0000.00I-1".EPL_FB_OUT_147_I2008_S94Out;
	Cyclic#1.::FBout.Array[148] AT %QW."8YFLM01.0000.00I-1".EPL_FB_OUT_148_I2008_S95Out;
	Cyclic#1.::FBout.Array[149] AT %QW."8YFLM01.0000.00I-1".EPL_FB_OUT_149_I2008_S96Out;
	Cyclic#1.::FBout.Array[15] AT %QW."8YFLM01.0000.00I-1".EPL_FB_OUT_15_I2008_S10Out;
	Cyclic#1.::FBout.Array[150] AT %QW."8YFLM01.0000.00I-1".EPL_FB_OUT_150_I2008_S97Out;
	Cyclic#1.::FBout.Array[151] AT %QW."8YFLM01.0000.00I-1".EPL_FB_OUT_151_I2008_S98Out;
	Cyclic#1.::FBout.Array[152] AT %QW."8YFLM01.0000.00I-1".EPL_FB_OUT_152_I2008_S99Out;
	Cyclic#1.::FBout.Array[153] AT %QW."8YFLM01.0000.00I-1".EPL_FB_OUT_153_I2008_S9AOut;
	Cyclic#1.::FBout.Array[154] AT %QW."8YFLM01.0000.00I-1".EPL_FB_OUT_154_I2008_S9BOut;
	Cyclic#1.::FBout.Array[155] AT %QW."8YFLM01.0000.00I-1".EPL_FB_OUT_155_I2008_S9COut;
	Cyclic#1.::FBout.Array[156] AT %QW."8YFLM01.0000.00I-1".EPL_FB_OUT_156_I2008_S9DOut;
	Cyclic#1.::FBout.Array[157] AT %QW."8YFLM01.0000.00I-1".EPL_FB_OUT_157_I2008_S9EOut;
	Cyclic#1.::FBout.Array[158] AT %QW."8YFLM01.0000.00I-1".EPL_FB_OUT_158_I2008_S9FOut;
	Cyclic#1.::FBout.Array[159] AT %QW."8YFLM01.0000.00I-1".EPL_FB_OUT_159_I2008_SA0Out;
	Cyclic#1.::FBout.Array[16] AT %QW."8YFLM01.0000.00I-1".EPL_FB_OUT_16_I2008_S11Out;
	Cyclic#1.::FBout.Array[160] AT %QW."8YFLM01.0000.00I-1".EPL_FB_OUT_160_I2008_SA1Out;
	Cyclic#1.::FBout.Array[161] AT %QW."8YFLM01.0000.00I-1".EPL_FB_OUT_161_I2008_SA2Out;
	Cyclic#1.::FBout.Array[162] AT %QW."8YFLM01.0000.00I-1".EPL_FB_OUT_162_I2008_SA3Out;
	Cyclic#1.::FBout.Array[163] AT %QW."8YFLM01.0000.00I-1".EPL_FB_OUT_163_I2008_SA4Out;
	Cyclic#1.::FBout.Array[164] AT %QW."8YFLM01.0000.00I-1".EPL_FB_OUT_164_I2008_SA5Out;
	Cyclic#1.::FBout.Array[165] AT %QW."8YFLM01.0000.00I-1".EPL_FB_OUT_165_I2008_SA6Out;
	Cyclic#1.::FBout.Array[166] AT %QW."8YFLM01.0000.00I-1".EPL_FB_OUT_166_I2008_SA7Out;
	Cyclic#1.::FBout.Array[167] AT %QW."8YFLM01.0000.00I-1".EPL_FB_OUT_167_I2008_SA8Out;
	Cyclic#1.::FBout.Array[168] AT %QW."8YFLM01.0000.00I-1".EPL_FB_OUT_168_I2008_SA9Out;
	Cyclic#1.::FBout.Array[169] AT %QW."8YFLM01.0000.00I-1".EPL_FB_OUT_169_I2008_SAAOut;
	Cyclic#1.::FBout.Array[17] AT %QW."8YFLM01.0000.00I-1".EPL_FB_OUT_17_I2008_S12Out;
	Cyclic#1.::FBout.Array[170] AT %QW."8YFLM01.0000.00I-1".EPL_FB_OUT_170_I2008_SABOut;
	Cyclic#1.::FBout.Array[171] AT %QW."8YFLM01.0000.00I-1".EPL_FB_OUT_171_I2008_SACOut;
	Cyclic#1.::FBout.Array[172] AT %QW."8YFLM01.0000.00I-1".EPL_FB_OUT_172_I2008_SADOut;
	Cyclic#1.::FBout.Array[173] AT %QW."8YFLM01.0000.00I-1".EPL_FB_OUT_173_I2008_SAEOut;
	Cyclic#1.::FBout.Array[174] AT %QW."8YFLM01.0000.00I-1".EPL_FB_OUT_174_I2008_SAFOut;
	Cyclic#1.::FBout.Array[175] AT %QW."8YFLM01.0000.00I-1".EPL_FB_OUT_175_I2008_SB0Out;
	Cyclic#1.::FBout.Array[176] AT %QW."8YFLM01.0000.00I-1".EPL_FB_OUT_176_I2008_SB1Out;
	Cyclic#1.::FBout.Array[177] AT %QW."8YFLM01.0000.00I-1".EPL_FB_OUT_177_I2008_SB2Out;
	Cyclic#1.::FBout.Array[178] AT %QW."8YFLM01.0000.00I-1".EPL_FB_OUT_178_I2008_SB3Out;
	Cyclic#1.::FBout.Array[179] AT %QW."8YFLM01.0000.00I-1".EPL_FB_OUT_179_I2008_SB4Out;
	Cyclic#1.::FBout.Array[18] AT %QW."8YFLM01.0000.00I-1".EPL_FB_OUT_18_I2008_S13Out;
	Cyclic#1.::FBout.Array[180] AT %QW."8YFLM01.0000.00I-1".EPL_FB_OUT_180_I2008_SB5Out;
	Cyclic#1.::FBout.Array[181] AT %QW."8YFLM01.0000.00I-1".EPL_FB_OUT_181_I2008_SB6Out;
	Cyclic#1.::FBout.Array[182] AT %QW."8YFLM01.0000.00I-1".EPL_FB_OUT_182_I2008_SB7Out;
	Cyclic#1.::FBout.Array[183] AT %QW."8YFLM01.0000.00I-1".EPL_FB_OUT_183_I2008_SB8Out;
	Cyclic#1.::FBout.Array[184] AT %QW."8YFLM01.0000.00I-1".EPL_FB_OUT_184_I2008_SB9Out;
	Cyclic#1.::FBout.Array[185] AT %QW."8YFLM01.0000.00I-1".EPL_FB_OUT_185_I2008_SBAOut;
	Cyclic#1.::FBout.Array[186] AT %QW."8YFLM01.0000.00I-1".EPL_FB_OUT_186_I2008_SBBOut;
	Cyclic#1.::FBout.Array[187] AT %QW."8YFLM01.0000.00I-1".EPL_FB_OUT_187_I2008_SBCOut;
	Cyclic#1.::FBout.Array[188] AT %QW."8YFLM01.0000.00I-1".EPL_FB_OUT_188_I2008_SBDOut;
	Cyclic#1.::FBout.Array[189] AT %QW."8YFLM01.0000.00I-1".EPL_FB_OUT_189_I2008_SBEOut;
	Cyclic#1.::FBout.Array[19] AT %QW."8YFLM01.0000.00I-1".EPL_FB_OUT_19_I2008_S14Out;
	Cyclic#1.::FBout.Array[190] AT %QW."8YFLM01.0000.00I-1".EPL_FB_OUT_190_I2008_SBFOut;
	Cyclic#1.::FBout.Array[191] AT %QW."8YFLM01.0000.00I-1".EPL_FB_OUT_191_I2008_SC0Out;
	Cyclic#1.::FBout.Array[192] AT %QW."8YFLM01.0000.00I-1".EPL_FB_OUT_192_I2008_SC1Out;
	Cyclic#1.::FBout.Array[193] AT %QW."8YFLM01.0000.00I-1".EPL_FB_OUT_193_I2008_SC2Out;
	Cyclic#1.::FBout.Array[194] AT %QW."8YFLM01.0000.00I-1".EPL_FB_OUT_194_I2008_SC3Out;
	Cyclic#1.::FBout.Array[195] AT %QW."8YFLM01.0000.00I-1".EPL_FB_OUT_195_I2008_SC4Out;
	Cyclic#1.::FBout.Array[196] AT %QW."8YFLM01.0000.00I-1".EPL_FB_OUT_196_I2008_SC5Out;
	Cyclic#1.::FBout.Array[197] AT %QW."8YFLM01.0000.00I-1".EPL_FB_OUT_197_I2008_SC6Out;
	Cyclic#1.::FBout.Array[198] AT %QW."8YFLM01.0000.00I-1".EPL_FB_OUT_198_I2008_SC7Out;
	Cyclic#1.::FBout.Array[199] AT %QW."8YFLM01.0000.00I-1".EPL_FB_OUT_199_I2008_SC8Out;
	Cyclic#1.::FBout.Array[2] AT %QW."8YFLM01.0000.00I-1".EPL_FB_OUT_2_I2008_S03Out;
	Cyclic#1.::FBout.Array[20] AT %QW."8YFLM01.0000.00I-1".EPL_FB_OUT_20_I2008_S15Out;
	Cyclic#1.::FBout.Array[21] AT %QW."8YFLM01.0000.00I-1".EPL_FB_OUT_21_I2008_S16Out;
	Cyclic#1.::FBout.Array[22] AT %QW."8YFLM01.0000.00I-1".EPL_FB_OUT_22_I2008_S17Out;
	Cyclic#1.::FBout.Array[23] AT %QW."8YFLM01.0000.00I-1".EPL_FB_OUT_23_I2008_S18Out;
	Cyclic#1.::FBout.Array[24] AT %QW."8YFLM01.0000.00I-1".EPL_FB_OUT_24_I2008_S19Out;
	Cyclic#1.::FBout.Array[25] AT %QW."8YFLM01.0000.00I-1".EPL_FB_OUT_25_I2008_S1AOut;
	Cyclic#1.::FBout.Array[26] AT %QW."8YFLM01.0000.00I-1".EPL_FB_OUT_26_I2008_S1BOut;
	Cyclic#1.::FBout.Array[27] AT %QW."8YFLM01.0000.00I-1".EPL_FB_OUT_27_I2008_S1COut;
	Cyclic#1.::FBout.Array[28] AT %QW."8YFLM01.0000.00I-1".EPL_FB_OUT_28_I2008_S1DOut;
	Cyclic#1.::FBout.Array[29] AT %QW."8YFLM01.0000.00I-1".EPL_FB_OUT_29_I2008_S1EOut;
	Cyclic#1.::FBout.Array[3] AT %QW."8YFLM01.0000.00I-1".EPL_FB_OUT_3_I2008_S04Out;
	Cyclic#1.::FBout.Array[30] AT %QW."8YFLM01.0000.00I-1".EPL_FB_OUT_30_I2008_S1FOut;
	Cyclic#1.::FBout.Array[31] AT %QW."8YFLM01.0000.00I-1".EPL_FB_OUT_31_I2008_S20Out;
	Cyclic#1.::FBout.Array[32] AT %QW."8YFLM01.0000.00I-1".EPL_FB_OUT_32_I2008_S21Out;
	Cyclic#1.::FBout.Array[33] AT %QW."8YFLM01.0000.00I-1".EPL_FB_OUT_33_I2008_S22Out;
	Cyclic#1.::FBout.Array[34] AT %QW."8YFLM01.0000.00I-1".EPL_FB_OUT_34_I2008_S23Out;
	Cyclic#1.::FBout.Array[35] AT %QW."8YFLM01.0000.00I-1".EPL_FB_OUT_35_I2008_S24Out;
	Cyclic#1.::FBout.Array[36] AT %QW."8YFLM01.0000.00I-1".EPL_FB_OUT_36_I2008_S25Out;
	Cyclic#1.::FBout.Array[37] AT %QW."8YFLM01.0000.00I-1".EPL_FB_OUT_37_I2008_S26Out;
	Cyclic#1.::FBout.Array[38] AT %QW."8YFLM01.0000.00I-1".EPL_FB_OUT_38_I2008_S27Out;
	Cyclic#1.::FBout.Array[39] AT %QW."8YFLM01.0000.00I-1".EPL_FB_OUT_39_I2008_S28Out;
	Cyclic#1.::FBout.Array[4] AT %QW."8YFLM01.0000.00I-1".EPL_FB_OUT_4_I2008_S05Out;
	Cyclic#1.::FBout.Array[40] AT %QW."8YFLM01.0000.00I-1".EPL_FB_OUT_40_I2008_S29Out;
	Cyclic#1.::FBout.Array[41] AT %QW."8YFLM01.0000.00I-1".EPL_FB_OUT_41_I2008_S2AOut;
	Cyclic#1.::FBout.Array[42] AT %QW."8YFLM01.0000.00I-1".EPL_FB_OUT_42_I2008_S2BOut;
	Cyclic#1.::FBout.Array[43] AT %QW."8YFLM01.0000.00I-1".EPL_FB_OUT_43_I2008_S2COut;
	Cyclic#1.::FBout.Array[44] AT %QW."8YFLM01.0000.00I-1".EPL_FB_OUT_44_I2008_S2DOut;
	Cyclic#1.::FBout.Array[45] AT %QW."8YFLM01.0000.00I-1".EPL_FB_OUT_45_I2008_S2EOut;
	Cyclic#1.::FBout.Array[46] AT %QW."8YFLM01.0000.00I-1".EPL_FB_OUT_46_I2008_S2FOut;
	Cyclic#1.::FBout.Array[47] AT %QW."8YFLM01.0000.00I-1".EPL_FB_OUT_47_I2008_S30Out;
	Cyclic#1.::FBout.Array[48] AT %QW."8YFLM01.0000.00I-1".EPL_FB_OUT_48_I2008_S31Out;
	Cyclic#1.::FBout.Array[49] AT %QW."8YFLM01.0000.00I-1".EPL_FB_OUT_49_I2008_S32Out;
	Cyclic#1.::FBout.Array[5] AT %QW."8YFLM01.0000.00I-1".EPL_FB_OUT_5_I2008_S06Out;
	Cyclic#1.::FBout.Array[50] AT %QW."8YFLM01.0000.00I-1".EPL_FB_OUT_50_I2008_S33Out;
	Cyclic#1.::FBout.Array[51] AT %QW."8YFLM01.0000.00I-1".EPL_FB_OUT_51_I2008_S34Out;
	Cyclic#1.::FBout.Array[52] AT %QW."8YFLM01.0000.00I-1".EPL_FB_OUT_52_I2008_S35Out;
	Cyclic#1.::FBout.Array[53] AT %QW."8YFLM01.0000.00I-1".EPL_FB_OUT_53_I2008_S36Out;
	Cyclic#1.::FBout.Array[54] AT %QW."8YFLM01.0000.00I-1".EPL_FB_OUT_54_I2008_S37Out;
	Cyclic#1.::FBout.Array[55] AT %QW."8YFLM01.0000.00I-1".EPL_FB_OUT_55_I2008_S38Out;
	Cyclic#1.::FBout.Array[56] AT %QW."8YFLM01.0000.00I-1".EPL_FB_OUT_56_I2008_S39Out;
	Cyclic#1.::FBout.Array[57] AT %QW."8YFLM01.0000.00I-1".EPL_FB_OUT_57_I2008_S3AOut;
	Cyclic#1.::FBout.Array[58] AT %QW."8YFLM01.0000.00I-1".EPL_FB_OUT_58_I2008_S3BOut;
	Cyclic#1.::FBout.Array[59] AT %QW."8YFLM01.0000.00I-1".EPL_FB_OUT_59_I2008_S3COut;
	Cyclic#1.::FBout.Array[6] AT %QW."8YFLM01.0000.00I-1".EPL_FB_OUT_6_I2008_S07Out;
	Cyclic#1.::FBout.Array[60] AT %QW."8YFLM01.0000.00I-1".EPL_FB_OUT_60_I2008_S3DOut;
	Cyclic#1.::FBout.Array[61] AT %QW."8YFLM01.0000.00I-1".EPL_FB_OUT_61_I2008_S3EOut;
	Cyclic#1.::FBout.Array[62] AT %QW."8YFLM01.0000.00I-1".EPL_FB_OUT_62_I2008_S3FOut;
	Cyclic#1.::FBout.Array[63] AT %QW."8YFLM01.0000.00I-1".EPL_FB_OUT_63_I2008_S40Out;
	Cyclic#1.::FBout.Array[64] AT %QW."8YFLM01.0000.00I-1".EPL_FB_OUT_64_I2008_S41Out;
	Cyclic#1.::FBout.Array[65] AT %QW."8YFLM01.0000.00I-1".EPL_FB_OUT_65_I2008_S42Out;
	Cyclic#1.::FBout.Array[66] AT %QW."8YFLM01.0000.00I-1".EPL_FB_OUT_66_I2008_S43Out;
	Cyclic#1.::FBout.Array[67] AT %QW."8YFLM01.0000.00I-1".EPL_FB_OUT_67_I2008_S44Out;
	Cyclic#1.::FBout.Array[68] AT %QW."8YFLM01.0000.00I-1".EPL_FB_OUT_68_I2008_S45Out;
	Cyclic#1.::FBout.Array[69] AT %QW."8YFLM01.0000.00I-1".EPL_FB_OUT_69_I2008_S46Out;
	Cyclic#1.::FBout.Array[7] AT %QW."8YFLM01.0000.00I-1".EPL_FB_OUT_7_I2008_S08Out;
	Cyclic#1.::FBout.Array[70] AT %QW."8YFLM01.0000.00I-1".EPL_FB_OUT_70_I2008_S47Out;
	Cyclic#1.::FBout.Array[71] AT %QW."8YFLM01.0000.00I-1".EPL_FB_OUT_71_I2008_S48Out;
	Cyclic#1.::FBout.Array[72] AT %QW."8YFLM01.0000.00I-1".EPL_FB_OUT_72_I2008_S49Out;
	Cyclic#1.::FBout.Array[73] AT %QW."8YFLM01.0000.00I-1".EPL_FB_OUT_73_I2008_S4AOut;
	Cyclic#1.::FBout.Array[74] AT %QW."8YFLM01.0000.00I-1".EPL_FB_OUT_74_I2008_S4BOut;
	Cyclic#1.::FBout.Array[75] AT %QW."8YFLM01.0000.00I-1".EPL_FB_OUT_75_I2008_S4COut;
	Cyclic#1.::FBout.Array[76] AT %QW."8YFLM01.0000.00I-1".EPL_FB_OUT_76_I2008_S4DOut;
	Cyclic#1.::FBout.Array[77] AT %QW."8YFLM01.0000.00I-1".EPL_FB_OUT_77_I2008_S4EOut;
	Cyclic#1.::FBout.Array[78] AT %QW."8YFLM01.0000.00I-1".EPL_FB_OUT_78_I2008_S4FOut;
	Cyclic#1.::FBout.Array[79] AT %QW."8YFLM01.0000.00I-1".EPL_FB_OUT_79_I2008_S50Out;
	Cyclic#1.::FBout.Array[8] AT %QW."8YFLM01.0000.00I-1".EPL_FB_OUT_8_I2008_S09Out;
	Cyclic#1.::FBout.Array[80] AT %QW."8YFLM01.0000.00I-1".EPL_FB_OUT_80_I2008_S51Out;
	Cyclic#1.::FBout.Array[81] AT %QW."8YFLM01.0000.00I-1".EPL_FB_OUT_81_I2008_S52Out;
	Cyclic#1.::FBout.Array[82] AT %QW."8YFLM01.0000.00I-1".EPL_FB_OUT_82_I2008_S53Out;
	Cyclic#1.::FBout.Array[83] AT %QW."8YFLM01.0000.00I-1".EPL_FB_OUT_83_I2008_S54Out;
	Cyclic#1.::FBout.Array[84] AT %QW."8YFLM01.0000.00I-1".EPL_FB_OUT_84_I2008_S55Out;
	Cyclic#1.::FBout.Array[85] AT %QW."8YFLM01.0000.00I-1".EPL_FB_OUT_85_I2008_S56Out;
	Cyclic#1.::FBout.Array[86] AT %QW."8YFLM01.0000.00I-1".EPL_FB_OUT_86_I2008_S57Out;
	Cyclic#1.::FBout.Array[87] AT %QW."8YFLM01.0000.00I-1".EPL_FB_OUT_87_I2008_S58Out;
	Cyclic#1.::FBout.Array[88] AT %QW."8YFLM01.0000.00I-1".EPL_FB_OUT_88_I2008_S59Out;
	Cyclic#1.::FBout.Array[89] AT %QW."8YFLM01.0000.00I-1".EPL_FB_OUT_89_I2008_S5AOut;
	Cyclic#1.::FBout.Array[9] AT %QW."8YFLM01.0000.00I-1".EPL_FB_OUT_9_I2008_S0AOut;
	Cyclic#1.::FBout.Array[90] AT %QW."8YFLM01.0000.00I-1".EPL_FB_OUT_90_I2008_S5BOut;
	Cyclic#1.::FBout.Array[91] AT %QW."8YFLM01.0000.00I-1".EPL_FB_OUT_91_I2008_S5COut;
	Cyclic#1.::FBout.Array[92] AT %QW."8YFLM01.0000.00I-1".EPL_FB_OUT_92_I2008_S5DOut;
	Cyclic#1.::FBout.Array[93] AT %QW."8YFLM01.0000.00I-1".EPL_FB_OUT_93_I2008_S5EOut;
	Cyclic#1.::FBout.Array[94] AT %QW."8YFLM01.0000.00I-1".EPL_FB_OUT_94_I2008_S5FOut;
	Cyclic#1.::FBout.Array[95] AT %QW."8YFLM01.0000.00I-1".EPL_FB_OUT_95_I2008_S60Out;
	Cyclic#1.::FBout.Array[96] AT %QW."8YFLM01.0000.00I-1".EPL_FB_OUT_96_I2008_S61Out;
	Cyclic#1.::FBout.Array[97] AT %QW."8YFLM01.0000.00I-1".EPL_FB_OUT_97_I2008_S62Out;
	Cyclic#1.::FBout.Array[98] AT %QW."8YFLM01.0000.00I-1".EPL_FB_OUT_98_I2008_S63Out;
	Cyclic#1.::FBout.Array[99] AT %QW."8YFLM01.0000.00I-1".EPL_FB_OUT_99_I2008_S64Out;
END_VAR
```

### Config_1.assembly6d - X20CP3586/mapp6D/Config_1.assembly6d
```
Element gAssembly6D_1 (Type=assembly6d)
  Simulation6D = SimOn
  Shuttles:
    MaxShuttleCount = 6
    ShuttleIDMode = RealTimeID
    DefaultPosition:
      DefZ = 1.0
      DefRx = 0
      DefRy = 0
      DefRz = 0
    Limits:
      InPlaneLimits:
        InPlaneVelLim = 1.0
        InPlaneAccLim = 10.0
        InPlaneEmergDec = 10.0
      ShortAxLim:
        ShortAxAccLim:
          AccZLim = 10.0
          AccRxLim = 10.0
          AccRyLim = 10.0
          AccRzLim = 10.0
        ShortAxVelLim:
          VelZLim = 0.15
          VelRxLim = 0.1
          VelRyLim = 0.1
          VelRzLim = 0.3
  CyclicChannel6D:
    ReadChannel:
      Xaxis = TRUE
      Yaxis = TRUE
      Zaxis = TRUE
      Rxaxis = TRUE
      Ryaxis = TRUE
      Rzaxis = TRUE
  Fieldbus6D:
    SyncMode6D = ExternalPlkSync
    NodeNumber = 16
  IOMapp:
    Input = ::FBin
    Output = ::FBout
  Layout:
    Layout6D[1] = Layout6D_1
```

### Config_2.layout6d - X20CP3586/mapp6D/Config_2.layout6d
```
Element Layout6D_1 (Type=layout6d)
  Segments:
    SegRow = 2
    SegCol = 2
    Segment[1]:
      X = 0
      Y = 0
      Name
      IsMaster = True
    Segment[2]:
      X = 0
      Y = 1
      Name
      IsMaster = False
    Segment[3]:
      X = 1
      Y = 0
      Name
      IsMaster = False
    Segment[4]:
      X = 1
      Y = 1
      Name
      IsMaster = False
```

## Logical view

Binary libraries used (declarations not repeated): operator, runtime, astime, AsIecCon, McBase, brsystem, AsBrStr, McAcp6D 1.00.0

### Global.typ - Global data types
```iecst
TYPE
	CtrlType : 	STRUCT
		Start : BOOL;
		Stop : BOOL;
		Reset : BOOL;
	END_STRUCT;
END_TYPE
```


### Program Logical/Program (IEC)

#### Variables.var
```iecst
VAR
	MC_BR_SegGetInfo_Acp6D_0 : MC_BR_SegGetInfo_Acp6D;
	GetSegment : BOOL;
	ShRef : {REDUND_UNREPLICABLE} Mc6DShuttleType;
	SegRef : Mc6DSegmentType;
	ZoneRef : Mc6DZoneType;
	GetZone : BOOL;
	MC_BR_AsmGetSegment_Acp6D_0 : MC_BR_AsmGetSegment_Acp6D;
	MC_BR_ShStop_Acp6D_0 : MC_BR_ShStop_Acp6D;
	MC_BR_ShRecover_Acp6D_0 : MC_BR_ShRecover_Acp6D;
	MC_BR_ShReadInfo_Acp6D_0 : MC_BR_ShReadInfo_Acp6D;
	MC_BR_ShLevitation_Acp6D_0 : MC_BR_ShLevitation_Acp6D;
	MC_BR_ShHalt_Acp6D_0 : MC_BR_ShHalt_Acp6D;
	MC_BR_ShBuffer_Acp6D_0 : MC_BR_ShBuffer_Acp6D;
	MC_BR_MoveShortAxis_Acp6D_0 : MC_BR_MoveShortAxis_Acp6D;
	MC_BR_MoveInPlane_Acp6D_0 : MC_BR_MoveInPlane_Acp6D;
	MC_BR_MoveArc_Acp6D_0 : MC_BR_MoveArc_Acp6D;
	MC_BR_Move6D_Acp6D_0 : MC_BR_Move6D_Acp6D;
	MC_BR_AsmStop_Acp6D_0 : MC_BR_AsmStop_Acp6D;
	MC_BR_AsmReboot_Acp6D_0 : MC_BR_AsmReboot_Acp6D;
	MC_BR_AsmReadStatus_Acp6D_0 : MC_BR_AsmReadStatus_Acp6D;
	MC_BR_AsmPowerOn_Acp6D_0 : MC_BR_AsmPowerOn_Acp6D;
	MC_BR_AsmPowerOff_Acp6D_0 : MC_BR_AsmPowerOff_Acp6D;
	MC_BR_AsmLevitation_Acp6D_0 : MC_BR_AsmLevitation_Acp6D;
	MC_BR_AsmHalt_Acp6D_0 : MC_BR_AsmHalt_Acp6D;
	MC_BR_AsmGetShuttle_Acp6D_0 : MC_BR_AsmGetShuttle_Acp6D;
	MC_BR_AsmGetInfo_Acp6D_0 : MC_BR_AsmGetInfo_Acp6D;
	MC_BR_AsmGetErrCode_Acp6D_0 : MC_BR_AsmGetErrCode_Acp6D;
	MC_BR_AsmBuffer_Acp6D_0 : MC_BR_AsmBuffer_Acp6D;
	GetShuttle : BOOL;
	GetAllShuttles : BOOL;
	i : USINT;
	MoveInPlaneAsync : BOOL;
	AllShRef : ARRAY[0..3] OF Mc6DShuttleType;
	MC_BR_AsmReset_Acp6D_0 : MC_BR_AsmReset_Acp6D;
	MC_BR_AsmReadInfo_Acp6D_0 : MC_BR_AsmReadInfo_Acp6D;
	MC_BR_ShStereotypeDefine_Acp6D_0 : MC_BR_ShStereotypeDefine_Acp6D;
	MC_BR_ShStereotypeAssign_Acp6D_0 : MC_BR_ShStereotypeAssign_Acp6D;
	MC_BR_ShStereotypeDelete_Acp6D_0 : MC_BR_ShStereotypeDelete_Acp6D;
	MC_BR_MoveCyclic_0 : MC_BR_MoveCyclicPosition_Acp6D;
	MC_BR_ReadCyclicPosition_0 : MC_BR_ReadCyclicPosition_Acp6D;
	MC_BR_ReadCyclicForce_0 : MC_BR_ReadCyclicForce_Acp6D;
	MC_BR_SegPowerOff_0 : MC_BR_SegPowerOff_Acp6D;
	MC_BR_SegPowerOn_0 : MC_BR_SegPowerOn_Acp6D;
	MC_BR_SegBarrierCommand_0 : MC_BR_SegBarrierCommand_Acp6D;
	MC_BR_SegGetBarrierInfo_0 : MC_BR_SegGetBarrierInfo_Acp6D;
	MC_BR_ZoneCreate_0 : MC_BR_ZoneCreate_Acp6D;
	MC_BR_AsmGetZone_0 : MC_BR_AsmGetZone_Acp6D;
	MC_BR_ZonePowerOff_0 : MC_BR_ZonePowerOff_Acp6D;
	MC_BR_ZonePowerOn_0 : MC_BR_ZonePowerOn_Acp6D;
	MC_BR_ZoneBarrierCommand_0 : MC_BR_ZoneBarrierCommand_Acp6D;
	MC_BR_ZoneGetBarrierInfo_0 : MC_BR_ZoneGetBarrierInfo_Acp6D;
	MC_BR_ShGetPayload_0 : MC_BR_ShGetPayload_Acp6D;
	MC_BR_MoveInPlaneAsync_0 : MC_BR_MoveInPlaneAsync_Acp6D;
	MoveSinus : BOOL;
	time : REAL;
	cycle_time : REAL;
	frequnecy : REAL;
	w : REAL;
	amplitude : REAL;
	Inc : REAL;
	setPosition : REAL;
END_VAR
VAR CONSTANT
	MAX_ENTRIES : UINT := 10000;
END_VAR
VAR
	errInc : UINT;
	ErrCmdIDOut : ARRAY[0..MAX_ENTRIES] OF UINT;
	ErrIDArr : ARRAY[0..MAX_ENTRIES] OF UINT;
END_VAR
```

#### Main.st
```iecst
PROGRAM _INIT
	MC_BR_AsmGetInfo_Acp6D_0.Assembly 		:= ADR(gAssembly6D_1);
	MC_BR_AsmGetShuttle_Acp6D_0.Assembly 	:= ADR(gAssembly6D_1);
	MC_BR_AsmPowerOn_Acp6D_0.Assembly 		:= ADR(gAssembly6D_1);
	MC_BR_AsmPowerOff_Acp6D_0.Assembly 		:= ADR(gAssembly6D_1);
	MC_BR_AsmReadStatus_Acp6D_0.Assembly 	:= ADR(gAssembly6D_1);
	MC_BR_AsmStop_Acp6D_0.Assembly			:= ADR(gAssembly6D_1);
	MC_BR_AsmHalt_Acp6D_0.Assembly			:= ADR(gAssembly6D_1);
	MC_BR_AsmLevitation_Acp6D_0.Assembly	:= ADR(gAssembly6D_1);
	MC_BR_AsmBuffer_Acp6D_0.Assembly		:= ADR(gAssembly6D_1);
	MC_BR_AsmReboot_Acp6D_0.Assembly		:= ADR(gAssembly6D_1);
	MC_BR_AsmGetErrCode_Acp6D_0.Assembly	:= ADR(gAssembly6D_1);
	MC_BR_AsmGetSegment_Acp6D_0.Assembly	:= ADR(gAssembly6D_1);
	MC_BR_AsmReset_Acp6D_0.Assembly			:= ADR(gAssembly6D_1);
	MC_BR_AsmReadInfo_Acp6D_0.Assembly			:= ADR(gAssembly6D_1);
	MC_BR_ShStereotypeDelete_Acp6D_0.Assembly		:= ADR(gAssembly6D_1);
	MC_BR_ZoneCreate_0.Assembly			:= ADR(gAssembly6D_1);
	MC_BR_ShStereotypeDefine_Acp6D_0.Assembly	:= ADR(gAssembly6D_1);
	MC_BR_AsmGetZone_0.Assembly				:= ADR(gAssembly6D_1);
	MC_BR_MoveInPlaneAsync_0.Assembly		:= ADR(gAssembly6D_1);

	FBin;
	FBout;

	cycle_time := 0.001;
	frequnecy := 1;
	amplitude := 1;
END_PROGRAM

PROGRAM _CYCLIC

	IF(GetShuttle)THEN
		MC_BR_AsmGetShuttle_Acp6D_0.Enable := TRUE;
		ShRef := MC_BR_AsmGetShuttle_Acp6D_0.Shuttle;
	ELSE
		MC_BR_AsmGetShuttle_Acp6D_0.Enable := FALSE;
	END_IF;

	IF(GetSegment)THEN
		MC_BR_AsmGetSegment_Acp6D_0.Enable := TRUE;
		SegRef := MC_BR_AsmGetSegment_Acp6D_0.Segment;
	ELSE
		MC_BR_AsmGetSegment_Acp6D_0.Enable	:= FALSE;
	END_IF;

	IF(GetAllShuttles)THEN
		MC_BR_AsmGetShuttle_Acp6D_0.Enable := TRUE;
		IF(MC_BR_AsmGetShuttle_Acp6D_0.Valid)THEN
			IF(MC_BR_AsmGetShuttle_Acp6D_0.Next)THEN
				AllShRef[i] := MC_BR_AsmGetShuttle_Acp6D_0.Shuttle;
				i := i+1;
				MC_BR_AsmGetShuttle_Acp6D_0.Next := FALSE;
			ELSE
				IF(i = 0)THEN
					AllShRef[i] := MC_BR_AsmGetShuttle_Acp6D_0.Shuttle;
					i := i+1;
				END_IF;

				MC_BR_AsmGetShuttle_Acp6D_0.Next := TRUE;
			END_IF;
		ELSIF(MC_BR_AsmGetShuttle_Acp6D_0.Error)THEN
			MC_BR_AsmGetShuttle_Acp6D_0.Enable := FALSE;
			GetAllShuttles := FALSE;
		END_IF;
	ELSE
		i := 0;
		//	MC_BR_AsmGetShuttle_Acp6D_0.Enable := FALSE;
	END_IF;

	IF(MoveInPlaneAsync)THEN
		MC_BR_MoveInPlaneAsync_0.Parameters.Acceleration := 10;
		MC_BR_MoveInPlaneAsync_0.Parameters.Velocity		:= 1;
		MC_BR_MoveInPlaneAsync_0.Parameters.AsyncPar[0].Shuttle := ADR(AllShRef[0]);
		MC_BR_MoveInPlaneAsync_0.Parameters.AsyncPar[0].X		:= 0.060;
		MC_BR_MoveInPlaneAsync_0.Parameters.AsyncPar[0].Y		:= 0.060;
		MC_BR_MoveInPlaneAsync_0.Execute := TRUE;
		IF(MC_BR_MoveInPlaneAsync_0.Done)THEN
			MC_BR_MoveInPlaneAsync_0.Execute := FALSE;
			MoveInPlaneAsync := FALSE;
		END_IF;
	END_IF;

	IF(GetZone)THEN
		MC_BR_AsmGetZone_0.Enable := TRUE;
		ZoneRef := MC_BR_AsmGetZone_0.Zone;
	ELSE
		MC_BR_AsmGetZone_0.Enable := FALSE;
	END_IF;

	MC_BR_ShReadInfo_Acp6D_0.Shuttle 	:= ADR(ShRef);
	MC_BR_MoveInPlane_Acp6D_0.Shuttle	:= ADR(ShRef);
	MC_BR_MoveShortAxis_Acp6D_0.Shuttle	:= ADR(ShRef);
	MC_BR_MoveArc_Acp6D_0.Shuttle		:= ADR(ShRef);
	MC_BR_ShLevitation_Acp6D_0.Shuttle	:= ADR(ShRef);
	MC_BR_Move6D_Acp6D_0.Shuttle		:= ADR(ShRef);
	MC_BR_ShBuffer_Acp6D_0.Shuttle		:= ADR(ShRef);
	MC_BR_ShStop_Acp6D_0.Shuttle		:= ADR(ShRef);
	MC_BR_ShHalt_Acp6D_0.Shuttle		:= ADR(ShRef);
	MC_BR_ShRecover_Acp6D_0.Shuttle		:= ADR(ShRef);
	MC_BR_MoveCyclic_0.Shuttle			:= ADR(ShRef);
	MC_BR_ShStereotypeAssign_Acp6D_0.Shuttle := ADR(ShRef);
	MC_BR_ReadCyclicPosition_0.Shuttle	:= ADR(ShRef);
	MC_BR_ReadCyclicForce_0.Shuttle		:= ADR(ShRef);
	MC_BR_ShGetPayload_0.Shuttle		:= ADR(ShRef);
	MC_BR_MoveInPlaneAsync_0.Parameters.AsyncPar[0].Shuttle := ADR(ShRef);
	MC_BR_MoveInPlaneAsync_0.Parameters.AsyncPar[0].X := 0.060;
	MC_BR_MoveInPlaneAsync_0.Parameters.AsyncPar[0].Y := 0.060;
	MC_BR_MoveInPlaneAsync_0.Parameters.Velocity := 1;
	MC_BR_MoveInPlaneAsync_0.Parameters.Acceleration := 10;

	MC_BR_SegGetInfo_Acp6D_0.Segment	:= ADR(SegRef);
	MC_BR_SegPowerOff_0.Segment			:= ADR(SegRef);
	MC_BR_SegPowerOn_0.Segment			:= ADR(SegRef);
	MC_BR_SegBarrierCommand_0.Segment	:= ADR(SegRef);
	MC_BR_SegGetBarrierInfo_0.Segment	:= ADR(SegRef);

	MC_BR_ZonePowerOff_0.Zone			:= ADR(ZoneRef);
	MC_BR_ZonePowerOn_0.Zone			:= ADR(ZoneRef);
	MC_BR_ZoneBarrierCommand_0.Zone		:= ADR(ZoneRef);
	MC_BR_ZoneGetBarrierInfo_0.Zone		:= ADR(ZoneRef);

//	IF(errInc <= MAX_ENTRIES)THEN
//		ErrIDArr[errInc] := FBin.Array[5];
//		ErrCmdIDOut[errInc] := FBout.Array[3];
//
//		errInc := errInc +1;
//	END_IF;

	MC_BR_SegGetInfo_Acp6D_0();
	MC_BR_AsmGetInfo_Acp6D_0();
	MC_BR_AsmGetShuttle_Acp6D_0();
	MC_BR_AsmPowerOn_Acp6D_0();
	MC_BR_AsmPowerOff_Acp6D_0();
	MC_BR_AsmReadStatus_Acp6D_0();
	MC_BR_ShReadInfo_Acp6D_0();
	MC_BR_MoveInPlane_Acp6D_0();
	MC_BR_MoveShortAxis_Acp6D_0();
	MC_BR_MoveArc_Acp6D_0();
	MC_BR_ShLevitation_Acp6D_0();
	MC_BR_Move6D_Acp6D_0();
	MC_BR_ShBuffer_Acp6D_0();
	MC_BR_ShStop_Acp6D_0();
	MC_BR_ShHalt_Acp6D_0();
	MC_BR_AsmStop_Acp6D_0();
	MC_BR_AsmHalt_Acp6D_0();
	MC_BR_AsmLevitation_Acp6D_0();
	MC_BR_AsmBuffer_Acp6D_0();
	MC_BR_ShRecover_Acp6D_0();
	MC_BR_AsmReboot_Acp6D_0();
	MC_BR_AsmGetErrCode_Acp6D_0();
	MC_BR_AsmGetSegment_Acp6D_0();
	MC_BR_AsmReset_Acp6D_0();
	MC_BR_AsmReadInfo_Acp6D_0();
	MC_BR_ShStereotypeAssign_Acp6D_0();
	MC_BR_ShStereotypeDefine_Acp6D_0();
	MC_BR_ShStereotypeDelete_Acp6D_0();
	MC_BR_MoveCyclic_0();
	MC_BR_ReadCyclicPosition_0();
	MC_BR_ReadCyclicForce_0();
	MC_BR_SegPowerOff_0();
	MC_BR_SegPowerOn_0();
	MC_BR_SegBarrierCommand_0();
	MC_BR_SegGetBarrierInfo_0();
	MC_BR_ZoneCreate_0();
	MC_BR_AsmGetZone_0();
	MC_BR_ZonePowerOff_0();
	MC_BR_ZonePowerOn_0();
	MC_BR_ZoneBarrierCommand_0();
	MC_BR_ZoneGetBarrierInfo_0();
	MC_BR_ShGetPayload_0();
	MC_BR_MoveInPlaneAsync_0();

END_PROGRAM

PROGRAM _EXIT
	(* Insert code here *)

END_PROGRAM
```

### Program Logical/Macro (IEC)

#### Main.st - Init, cyclic, exit code
```iecst
PROGRAM _INIT
	(* Insert code here *)

	MacroName := 'TestMacro';
	inc			:= 0;
	MC_BR_MacroCreate_Acp6D_0.Assembly := ADR(gAssembly6D_1);
	MC_BR_AsmPowerOn_Acp6D_0.Assembly	:= ADR(gAssembly6D_1);
	MC_BR_AsmReadStatus_0.Assembly		:= ADR(gAssembly6D_1);
	MC_BR_MacroDelete_0.Assembly		:= ADR(gAssembly6D_1);
	MC_BR_AsmGetShuttle_0.Assembly		:= ADR(gAssembly6D_1);
END_PROGRAM

PROGRAM _CYCLIC
	CASE MacroState OF
		0:
			ResetMacroFubs;
			IF(Cmd.Start)THEN
				MacroState := MacroState+1;
				MC_BR_AsmReadStatus_0.Enable := TRUE;
			END_IF;

		1:
			IF(MC_BR_AsmReadStatus_0.Valid)THEN
				IF(MC_BR_AsmReadStatus_0.AssemblyDisabled)THEN
					MacroState := MacroState+1;
				ELSIF(MC_BR_AsmReadStatus_0.AssemblyReady)THEN
					MacroState := MacroState+2;
				END_IF;
			END_IF;

		2:
			MC_BR_AsmPowerOn_Acp6D_0.Execute := TRUE;
			IF(MC_BR_AsmPowerOn_Acp6D_0.Done)THEN
				MC_BR_AsmPowerOn_Acp6D_0.Execute := FALSE;
				MacroState := MacroState+1;
			END_IF;

		3:
			MC_BR_MacroCreate_Acp6D_0.Parameters.Name := MacroName;
			int_to_str := USINT_TO_STRING(inc);
			brsstrcat(ADR(MC_BR_MacroCreate_Acp6D_0.Parameters.Name),ADR(int_to_str));
			TempName := MC_BR_MacroCreate_Acp6D_0.Parameters.Name;
			MC_BR_MacroCreate_Acp6D_0.Execute := TRUE;

			IF(MC_BR_MacroCreate_Acp6D_0.Done)THEN
				inc := inc+1;
				MacroSh := MC_BR_MacroCreate_Acp6D_0.MacroShuttle;
				MC_BR_MacroCreate_Acp6D_0.Execute := FALSE;
				MacroState := MacroState+1;
			END_IF;

		4:
			MC_BR_MoveInPlane_Acp6D_0.Shuttle := ADR(MacroSh);
			MC_BR_MoveInPlane_Acp6D_0.Parameters.Acceleration := 10;
			MC_BR_MoveInPlane_Acp6D_0.Parameters.Velocity	:= 1;
			MC_BR_MoveInPlane_Acp6D_0.Parameters.Mode		:= 1;
			MC_BR_MoveInPlane_Acp6D_0.Parameters.Path		:= 0;
			MC_BR_MoveInPlane_Acp6D_0.Parameters.Position.X := 0.120;
			MC_BR_MoveInPlane_Acp6D_0.Parameters.Position.Y	:= 0;
			MC_BR_MoveInPlane_Acp6D_0.Execute := TRUE;

			IF(MC_BR_MoveInPlane_Acp6D_0.Acknowledge)THEN
				MC_BR_MoveInPlane_Acp6D_0.Execute := FALSE;
				MacroState := MacroState+1;
			END_IF;
		5:
			//	IF(MC_BR_MoveInPlane_Acp6D_0.Acknowledge = FALSE)THEN
			MC_BR_MoveInPlane_Acp6D_0.Shuttle := ADR(MacroSh);
			MC_BR_MoveInPlane_Acp6D_0.Parameters.Acceleration := 10;
			MC_BR_MoveInPlane_Acp6D_0.Parameters.Velocity	:= 1;
			MC_BR_MoveInPlane_Acp6D_0.Parameters.Mode		:= 1;
			MC_BR_MoveInPlane_Acp6D_0.Parameters.Path		:= 0;
			MC_BR_MoveInPlane_Acp6D_0.Parameters.Position.X := -0.120;
			MC_BR_MoveInPlane_Acp6D_0.Parameters.Position.Y	:= 0;
			MC_BR_MoveInPlane_Acp6D_0.Execute := TRUE;
			//END_IF;

			IF(MC_BR_MoveInPlane_Acp6D_0.Acknowledge)THEN
				MC_BR_MoveInPlane_Acp6D_0.Execute := FALSE;
				IF(Clear)THEN
					MacroState := MacroState+2;
				ELSE
					MacroState := MacroState+1;
				END_IF;
			END_IF;

		6:
			MC_BR_MacroSave_0.Shuttle := ADR(MacroSh);
			MC_BR_MacroSave_0.Execute := TRUE;
			IF(MC_BR_MacroSave_0.Done)THEN
				MC_BR_MacroSave_0.Execute := FALSE;
				MacroState := MacroState+1;
				i := 0;
			ELSIF(MC_BR_MacroSave_0.Error AND Clear)THEN
				MC_BR_MacroSave_0.Execute := FALSE;
				MacroState := 10;
			END_IF;

		7:
			MC_BR_AsmGetShuttle_0.Enable := TRUE;
			IF(MC_BR_AsmGetShuttle_0.Valid)THEN
				IF(MC_BR_AsmGetShuttle_0.Next)THEN
					ShRefArr[i] := MC_BR_AsmGetShuttle_0.Shuttle;
					i := i+1;
					MC_BR_AsmGetShuttle_0.Next := FALSE;
				ELSE
					IF(i = 0)THEN
						ShRefArr[i] := MC_BR_AsmGetShuttle_0.Shuttle;
						i := i+1;
					END_IF;

					MC_BR_AsmGetShuttle_0.Next := TRUE;
				END_IF;
			ELSIF(MC_BR_AsmGetShuttle_0.Error)THEN
				MC_BR_AsmGetShuttle_0.Enable := FALSE;
				MacroState := MacroState+1;
			END_IF;

		8:
			MC_BR_MacroRun_0.Shuttle := ADR(ShRefArr[0]);
			MC_BR_MacroRun_0.Execute := TRUE;
			MC_BR_MacroRun_0.Name	:= TempName;

			IF(MC_BR_MacroRun_0.Done)THEN
				MC_BR_MacroRun_0.Execute := FALSE;
				MacroState := MacroState+1;
			END_IF;

		9:
			MC_BR_MacroClear_0.Shuttle := ADR(MacroSh);
			MC_BR_MacroClear_0.Execute := TRUE;
			IF(MC_BR_MacroClear_0.Done)THEN
				MC_BR_MacroClear_0.Execute := FALSE;
				MacroState := 6;
			END_IF;

		10:
			IF(Cmd.Reset)THEN
				MacroState := 0;
				Cmd.Start := FALSE;
				Cmd.Reset := FALSE;
				Cmd.Stop := FALSE;
				Clear := FALSE;
			END_IF;

	END_CASE;

	MC_BR_AsmPowerOn_Acp6D_0();
	MC_BR_MacroCreate_Acp6D_0();
	MC_BR_MoveInPlane_Acp6D_0();
	MC_BR_AsmReadStatus_0();
	MC_BR_MacroSave_0();
	MC_BR_MacroClear_0();
	MC_BR_MacroDelete_0();
	MC_BR_MacroRun_0();
	MC_BR_AsmGetShuttle_0();
END_PROGRAM

PROGRAM _EXIT
	(* Insert code here *)

END_PROGRAM
```

#### Variables.var - Local variables
```iecst
VAR
	MC_BR_AsmPowerOn_Acp6D_0 : MC_BR_AsmPowerOn_Acp6D;
	MC_BR_MacroCreate_Acp6D_0 : MC_BR_MacroCreate_Acp6D;
	MC_BR_MoveInPlane_Acp6D_0 : MC_BR_MoveInPlane_Acp6D;
	MacroSh : {REDUND_UNREPLICABLE} Mc6DShuttleType;
	MacroState : USINT;
	Cmd : CtrlType;
	MacroName : STRING[28];
	inc : USINT;
	helpStr : STRING[28];
	int_to_str : STRING[4];
	MC_BR_AsmReadStatus_0 : MC_BR_AsmReadStatus_Acp6D;
	MC_BR_MacroSave_0 : MC_BR_MacroSave_Acp6D;
	MC_BR_MacroClear_0 : MC_BR_MacroClear_Acp6D;
	Clear : BOOL;
	MC_BR_MacroDelete_0 : MC_BR_MacroDelete_Acp6D;
	MC_BR_MacroRun_0 : MC_BR_MacroRun_Acp6D;
	MC_BR_AsmGetShuttle_0 : MC_BR_AsmGetShuttle_Acp6D;
	ShRefArr : ARRAY[0..MAX_NUM_SH] OF Mc6DShuttleType;
END_VAR
VAR CONSTANT
	MAX_NUM_SH : USINT := 10;
END_VAR
VAR
	i : USINT;
	TempName : STRING[33];
END_VAR
```

#### ResetMacroFubs.st
```iecst
ACTION ResetMacroFubs:

	MC_BR_MacroCreate_Acp6D_0.Execute := FALSE;
	MC_BR_MoveInPlane_Acp6D_0.Execute := FALSE;
	MC_BR_AsmPowerOn_Acp6D_0.Execute := FALSE;

END_ACTION
```

### Program Logical/ShuttleGroup (IEC)

#### Main.st - Init, cyclic, exit code
```iecst
PROGRAM _INIT
	MC_BR_ShGroupCreate_0.Assembly := ADR(gAssembly6D_1);
	MC_BR_AsmPowerOn_Acp6D_0.Assembly	:= ADR(gAssembly6D_1);
	MC_BR_AsmReadStatus_0.Assembly		:= ADR(gAssembly6D_1);
	MC_BR_AsmGetShuttle_0.Assembly		:= ADR(gAssembly6D_1);
	MC_BR_AsmGetShGroup_0.Assembly		:= ADR(gAssembly6D_1);
	ShGroupState := 0;
END_PROGRAM

PROGRAM _CYCLIC
	CASE ShGroupState OF
		0:
			ResetShGroupFubs;
			IF(Cmd.Start)THEN
				ShGroupState := ShGroupState+1;
				MC_BR_AsmReadStatus_0.Enable := TRUE;
			END_IF;

		1:
			IF(MC_BR_AsmReadStatus_0.Valid)THEN
				IF(MC_BR_AsmReadStatus_0.AssemblyDisabled)THEN
					ShGroupState := ShGroupState+1;
				ELSIF(MC_BR_AsmReadStatus_0.AssemblyReady)THEN
					ShGroupState := ShGroupState+2;
				END_IF;
			END_IF;

		2:
			MC_BR_AsmPowerOn_Acp6D_0.Execute := TRUE;
			IF(MC_BR_AsmPowerOn_Acp6D_0.Done)THEN
				MC_BR_AsmPowerOn_Acp6D_0.Execute := FALSE;
				ShGroupState := ShGroupState+1;
			END_IF;

		3:
			MC_BR_ShGroupCreate_0.Execute := TRUE;

			IF(MC_BR_ShGroupCreate_0.Done)THEN
				ShGroupRef := MC_BR_ShGroupCreate_0.ShuttleGroup;
				MC_BR_ShGroupCreate_0.Execute := FALSE;
				ShGroupState := ShGroupState+1;
				i := 0;
			END_IF;

		4:
			MC_BR_AsmGetShuttle_0.Enable := TRUE;
			IF(MC_BR_AsmGetShuttle_0.Valid)THEN
				IF(MC_BR_AsmGetShuttle_0.Next)THEN
					ShRefArr[i] := MC_BR_AsmGetShuttle_0.Shuttle;
					i := i+1;
					MC_BR_AsmGetShuttle_0.Next := FALSE;
				ELSE
					IF(i = 0)THEN
						ShRefArr[i] := MC_BR_AsmGetShuttle_0.Shuttle;
						i := i+1;
					END_IF;

					MC_BR_AsmGetShuttle_0.Next := TRUE;
				END_IF;
			ELSIF(MC_BR_AsmGetShuttle_0.Error)THEN
				MC_BR_AsmGetShuttle_0.Enable := FALSE;
				ShGroupState := ShGroupState+1;
			END_IF;

		5:
			MC_BR_ShGroupAddShuttle_0.ShuttleGroup := ADR(ShGroupRef);
			FOR i := 0 TO MAX_NUM_SH BY 1 DO
				IF(ShRefArr[i].controlif>0)THEN
					MC_BR_ShGroupAddShuttle_0.Parameters.ShuttleList[i].Shuttle := ADR(ShRefArr[i]);
				END_IF;
			END_FOR;
			MC_BR_ShGroupAddShuttle_0.Execute := TRUE;

			IF(MC_BR_ShGroupAddShuttle_0.Done)THEN
				MC_BR_ShGroupAddShuttle_0.Execute := FALSE;
				ShGroupState := ShGroupState+1;
			END_IF;

		6:
			IF(Cmd.Reset)THEN
				ShGroupState := 0;
				Cmd.Start := FALSE;
				Cmd.Reset := FALSE;
				Cmd.Stop := FALSE;
			END_IF;

	END_CASE;

	MC_BR_ShGroupClear_0.ShuttleGroup 		:= ADR(ShGroupRef);
	MC_BR_ShGroupGetInfo_0.ShuttleGroup	:= ADR(ShGroupRef);
	MC_BR_ShGroupCoupleCtrl_0.ShuttleGroup	:= ADR(ShGroupRef);
	MC_BR_ShGroupBuffer_0.ShuttleGroup		:= ADR(ShGroupRef);
	MC_BR_ShGroupDelete_0.ShuttleGroup		:= ADR(ShGroupRef);

	MC_BR_ShGroupDelete_0();
	MC_BR_AsmGetShGroup_0();
	MC_BR_ShGroupBuffer_0();
	MC_BR_ShGroupCoupleCtrl_0();
	MC_BR_ShGroupGetInfo_0();
	MC_BR_ShGroupClear_0();
	MC_BR_ShGroupAddShuttle_0();
	MC_BR_AsmGetShuttle_0();
	MC_BR_ShGroupCreate_0();
	MC_BR_AsmReadStatus_0();
	MC_BR_AsmPowerOn_Acp6D_0();

END_PROGRAM

PROGRAM _EXIT
	(* Insert code here *)

END_PROGRAM
```

#### Variables.var - Local variables
```iecst
VAR
	MC_BR_ShGroupCreate_0 : MC_BR_ShGroupCreate_Acp6D;
	MC_BR_AsmPowerOn_Acp6D_0 : MC_BR_AsmPowerOn_Acp6D;
	MC_BR_AsmReadStatus_0 : MC_BR_AsmReadStatus_Acp6D;
	Cmd : CtrlType;
	ShGroupState : USINT;
	ShGroupRef : Mc6DShuttleGroupType;
	MC_BR_ShGroupAddShuttle_0 : MC_BR_ShGroupAddShuttle_Acp6D;
	MC_BR_AsmGetShuttle_0 : MC_BR_AsmGetShuttle_Acp6D;
	ShRefArr : ARRAY[0..MAX_NUM_SH] OF Mc6DShuttleType;
END_VAR
VAR CONSTANT
	MAX_NUM_SH : USINT := 10;
END_VAR
VAR
	i : USINT;
	MC_BR_ShGroupClear_0 : MC_BR_ShGroupClear_Acp6D;
	MC_BR_ShGroupGetInfo_0 : MC_BR_ShGroupGetInfo_Acp6D;
	MC_BR_ShGroupCoupleCtrl_0 : MC_BR_ShGroupCoupleCtrl_Acp6D;
	MC_BR_ShGroupBuffer_0 : MC_BR_ShGroupBuffer_Acp6D;
	MC_BR_AsmGetShGroup_0 : MC_BR_AsmGetShGroup_Acp6D;
	MC_BR_ShGroupDelete_0 : MC_BR_ShGroupDelete_Acp6D;
END_VAR
```

#### ResetShGroupFubs.st
```iecst
ACTION ResetShGroupFubs:
	MC_BR_ShGroupCreate_0.Execute := FALSE;
	MC_BR_AsmPowerOn_Acp6D_0.Execute := FALSE;

END_ACTION
```

### Program Logical/VirtualShuttle1 (IEC)

#### Main.st - Init, cyclic, exit code
```iecst
PROGRAM _INIT
	MC_BR_AsmPowerOn_Acp6D_0.Assembly	:= ADR(gAssembly6D_1);
	MC_BR_AsmReadStatus_0.Assembly		:= ADR(gAssembly6D_1);
	MC_BR_AsmGetVirtualSh_0.Assembly		:= ADR(gAssembly6D_1);
	MC_BR_VirtualShCreate_0.Assembly	:= ADR(gAssembly6D_1);
	MC_BR_AsmGetVirtualSh_0.Assembly	:= ADR(gAssembly6D_1);
	VirtualShState := 0;
END_PROGRAM

PROGRAM _CYCLIC
	CASE VirtualShState OF
		0:
			ResetShGroupFubs;
			IF(Cmd.Start)THEN
				VirtualShState := VirtualShState+1;
				MC_BR_AsmReadStatus_0.Enable := TRUE;
			END_IF;

		1:
			IF(MC_BR_AsmReadStatus_0.Valid)THEN
				IF(MC_BR_AsmReadStatus_0.AssemblyDisabled)THEN
					VirtualShState := VirtualShState+1;
				ELSIF(MC_BR_AsmReadStatus_0.AssemblyReady)THEN
					VirtualShState := VirtualShState+2;
				END_IF;
			END_IF;

		2:
			MC_BR_AsmPowerOn_Acp6D_0.Execute := TRUE;
			IF(MC_BR_AsmPowerOn_Acp6D_0.Done)THEN
				MC_BR_AsmPowerOn_Acp6D_0.Execute := FALSE;
				VirtualShState := VirtualShState+1;
			END_IF;

		3:
			MC_BR_VirtualShCreate_0.Execute := TRUE;

			IF(MC_BR_VirtualShCreate_0.Done)THEN
				VirtualShRef := MC_BR_VirtualShCreate_0.VirtualShuttle;
				MC_BR_VirtualShCreate_0.Execute := FALSE;
				VirtualShState := VirtualShState+1;
				i := 0;
			END_IF;

		4:
			MC_BR_AsmGetVirtualSh_0.Enable := TRUE;
			IF(MC_BR_AsmGetVirtualSh_0.Valid)THEN
				IF(MC_BR_AsmGetVirtualSh_0.Next)THEN
					VirtualShRefArr[i] := MC_BR_AsmGetVirtualSh_0.VirtualShuttle;
					i := i+1;
					MC_BR_AsmGetVirtualSh_0.Next := FALSE;
				ELSE
					IF(i = 0)THEN
						VirtualShRefArr[i] := MC_BR_AsmGetVirtualSh_0.VirtualShuttle;
						i := i+1;
					END_IF;

					MC_BR_AsmGetVirtualSh_0.Next := TRUE;
				END_IF;
			ELSIF(MC_BR_AsmGetVirtualSh_0.Error)THEN
				MC_BR_AsmGetVirtualSh_0.Enable := FALSE;
				VirtualShState := VirtualShState+1;
			END_IF;

		5:
			MC_BR_MoveInPlane_0.Shuttle := ADR(VirtualShRef);
			MC_BR_MoveInPlane_0.Parameters.Acceleration := 10;
			MC_BR_MoveInPlane_0.Parameters.Velocity := 1;
			MC_BR_MoveInPlane_0.Parameters.EndVelocity := 0;
			MC_BR_MoveInPlane_0.Parameters.Mode := 1;
			MC_BR_MoveInPlane_0.Parameters.Path := 0;
			MC_BR_MoveInPlane_0.Parameters.Position.X := 0.12;
			MC_BR_MoveInPlane_0.Parameters.Position.Y := 0.12;
			MC_BR_MoveInPlane_0.Execute := TRUE;

			IF(MC_BR_MoveInPlane_0.Acknowledge)THEN
				MC_BR_MoveInPlane_0.Execute := FALSE;
				VirtualShState := VirtualShState+1;
			END_IF;
		6:
			IF(Cmd.Reset)THEN
				VirtualShState := 0;
				Cmd.Start := FALSE;
				Cmd.Reset := FALSE;
				Cmd.Stop := FALSE;
			END_IF;

	END_CASE;

	MC_BR_MoveInPlane_0();
	MC_BR_AsmGetVirtualSh_0();
	MC_BR_VirtualShCreate_0();
	MC_BR_AsmReadStatus_0();
	MC_BR_AsmPowerOn_Acp6D_0();

END_PROGRAM

PROGRAM _EXIT
	(* Insert code here *)

END_PROGRAM
```

#### Variables.var - Local variables
```iecst
VAR
	MC_BR_ShGroupCreate_0 : MC_BR_ShGroupCreate_Acp6D;
	MC_BR_AsmPowerOn_Acp6D_0 : MC_BR_AsmPowerOn_Acp6D;
	MC_BR_AsmReadStatus_0 : MC_BR_AsmReadStatus_Acp6D;
	Cmd : CtrlType;
	VirtualShState : USINT;
	VirtualShRef : Mc6DShuttleGroupType;
	MC_BR_ShGroupAddShuttle_0 : MC_BR_ShGroupAddShuttle_Acp6D;
	MC_BR_AsmGetShuttle_0 : MC_BR_AsmGetShuttle_Acp6D;
	VirtualShRefArr : ARRAY[0..MAX_NUM_SH] OF Mc6DShuttleType;
END_VAR
VAR CONSTANT
	MAX_NUM_SH : USINT := 10;
END_VAR
VAR
	i : USINT;
	MC_BR_AsmGetVirtualSh_0 : MC_BR_AsmGetVirtualSh_Acp6D;
	MC_BR_VirtualShCreate_0 : MC_BR_VirtualShCreate_Acp6D;
	MC_BR_MoveInPlane_0 : MC_BR_MoveInPlane_Acp6D;
END_VAR
```

#### ResetVShFubs.st
```iecst
ACTION ResetShGroupFubs:
	MC_BR_AsmPowerOn_Acp6D_0.Execute := FALSE;
	MC_BR_VirtualShCreate_0.Execute := FALSE;

END_ACTION
```

### Program Logical/Planet (IEC)

#### Main.st - Init, cyclic, exit code
```iecst
PROGRAM _INIT
	MC_BR_AsmPowerOn_Acp6D_0.Assembly	:= ADR(gAssembly6D_1);
	MC_BR_AsmReadStatus_0.Assembly		:= ADR(gAssembly6D_1);
	MC_BR_AsmGetVirtualSh_0.Assembly		:= ADR(gAssembly6D_1);
	MC_BR_VirtualShCreate_0.Assembly	:= ADR(gAssembly6D_1);
	MC_BR_AsmGetVirtualSh_0.Assembly	:= ADR(gAssembly6D_1);
	MC_BR_AsmGetShuttle_0.Assembly		:= ADR(gAssembly6D_1);
	PlanetState := 0;
END_PROGRAM

PROGRAM _CYCLIC
	CASE PlanetState OF
		0:
			ResetPlanetFub;
			IF(Cmd.Start)THEN
				PlanetState := PlanetState+1;
				MC_BR_AsmReadStatus_0.Enable := TRUE;
			END_IF;

		1:
			IF(MC_BR_AsmReadStatus_0.Valid)THEN
				IF(MC_BR_AsmReadStatus_0.AssemblyDisabled)THEN
					PlanetState := PlanetState+1;
				ELSIF(MC_BR_AsmReadStatus_0.AssemblyReady)THEN
					PlanetState := PlanetState+2;
				END_IF;
			END_IF;

		2:
			MC_BR_AsmPowerOn_Acp6D_0.Execute := TRUE;
			IF(MC_BR_AsmPowerOn_Acp6D_0.Done)THEN
				MC_BR_AsmPowerOn_Acp6D_0.Execute := FALSE;
				PlanetState := PlanetState+1;
			END_IF;

		3:
			MC_BR_VirtualShCreate_0.Execute := TRUE;

			IF(MC_BR_VirtualShCreate_0.Done)THEN
				VirtualShRef := MC_BR_VirtualShCreate_0.VirtualShuttle;
				MC_BR_VirtualShCreate_0.Execute := FALSE;
				PlanetState := PlanetState+1;
				i := 0;
			END_IF;

		4:
			MC_BR_AsmGetShuttle_0.Enable := TRUE;
			IF(MC_BR_AsmGetShuttle_0.Valid)THEN
				IF(MC_BR_AsmGetShuttle_0.Next)THEN
					PlanetShRefArr[i] := MC_BR_AsmGetShuttle_0.Shuttle;
					i := i+1;
					MC_BR_AsmGetShuttle_0.Next := FALSE;
				ELSE
					IF(i = 0)THEN
						PlanetShRefArr[i] := MC_BR_AsmGetShuttle_0.Shuttle;
						i := i+1;
					END_IF;

					MC_BR_AsmGetShuttle_0.Next := TRUE;
				END_IF;
			ELSIF(MC_BR_AsmGetShuttle_0.Error)THEN
				MC_BR_AsmGetShuttle_0.Enable := FALSE;
				PlanetState := PlanetState+1;
			END_IF;

		5:
			MC_BR_ShPlanet_0.Shuttle := ADR(VirtualShRef);
			MC_BR_ShPlanet_0.Parameters.ShuttleList[0].Shuttle := ADR(PlanetShRefArr[0]);
			MC_BR_ShPlanet_0.Parameters.ShuttleList[1].Shuttle := ADR(PlanetShRefArr[1]);
			MC_BR_ShPlanet_0.Parameters.Option				   := mcACP6D_PLANET_ADD_SH;
			MC_BR_ShPlanet_0.Execute := TRUE;

			IF(MC_BR_ShPlanet_0.Done)THEN
				MC_BR_ShPlanet_0.Execute := FALSE;
				PlanetState := PlanetState +1;
			END_IF;

		6:
			MC_BR_MoveInPlane_0.Shuttle := ADR(VirtualShRef);
			MC_BR_MoveInPlane_0.Parameters.Acceleration := 10;
			MC_BR_MoveInPlane_0.Parameters.Velocity := 1;
			MC_BR_MoveInPlane_0.Parameters.EndVelocity := 0;
			MC_BR_MoveInPlane_0.Parameters.Mode := 1;
			MC_BR_MoveInPlane_0.Parameters.Path := 0;
			MC_BR_MoveInPlane_0.Parameters.Position.X := 0.12;
			MC_BR_MoveInPlane_0.Parameters.Position.Y := 0.12;
			MC_BR_MoveInPlane_0.Execute := TRUE;

			IF(MC_BR_MoveInPlane_0.Acknowledge)THEN
				MC_BR_MoveInPlane_0.Execute := FALSE;
				PlanetState := PlanetState+1;
			END_IF;
		7:
			IF(Cmd.Reset)THEN
				PlanetState := 0;
				Cmd.Start := FALSE;
				Cmd.Reset := FALSE;
				Cmd.Stop := FALSE;
			END_IF;

	END_CASE;

	MC_BR_MoveInPlane_0();
	MC_BR_AsmGetShuttle_0();
	MC_BR_VirtualShCreate_0();
	MC_BR_AsmReadStatus_0();
	MC_BR_AsmPowerOn_Acp6D_0();
	MC_BR_ShPlanet_0();

END_PROGRAM

PROGRAM _EXIT
	(* Insert code here *)

END_PROGRAM
```

#### Variables.var - Local variables
```iecst
VAR
	MC_BR_ShGroupCreate_0 : MC_BR_ShGroupCreate_Acp6D;
	MC_BR_AsmPowerOn_Acp6D_0 : MC_BR_AsmPowerOn_Acp6D;
	MC_BR_AsmReadStatus_0 : MC_BR_AsmReadStatus_Acp6D;
	Cmd : CtrlType;
	PlanetState : USINT;
	VirtualShRef : Mc6DShuttleGroupType;
	MC_BR_AsmGetShuttle_0 : MC_BR_AsmGetShuttle_Acp6D;
	PlanetShRefArr : ARRAY[0..MAX_NUM_SH] OF Mc6DShuttleType;
END_VAR
VAR CONSTANT
	MAX_NUM_SH : USINT := 10;
END_VAR
VAR
	i : USINT;
	MC_BR_VirtualShCreate_0 : MC_BR_VirtualShCreate_Acp6D;
	MC_BR_AsmGetVirtualSh_0 : MC_BR_AsmGetVirtualSh_Acp6D;
	MC_BR_MoveInPlane_0 : MC_BR_MoveInPlane_Acp6D;
	MC_BR_ShPlanet_0 : MC_BR_ShPlanet_Acp6D;
END_VAR
```

#### PlanetFub.st
```iecst
ACTION ResetPlanetFub:
	MC_BR_AsmPowerOn_Acp6D_0.Execute 	:= FALSE;
	MC_BR_VirtualShCreate_0.Execute 	:= FALSE;
	MC_BR_ShPlanet_0.Execute			:= FALSE;

END_ACTION
```

Listed in the project but not available here: Logical/Global.var, Logical/Macro/Types.typ, Logical/ShuttleGroup/Types.typ, Logical/VirtualShuttle1/Types.typ, Logical/Planet/Types.typ
